// TwinCAT 3 PLC project PLC
// ProgramVersion: 3.1.4026.13
// CompilerDefines: VISU_USEPROPERTYINFO
// libraries:
//   Tc2_Standard, * (Beckhoff Automation GmbH)
//   Tc2_System, * (Beckhoff Automation GmbH)
//   VisuSymbols, 4.5.0.0 (System)
// project tree:
//   FBs/Control/Function Blocks/ FB_Config.TcPOU, FB_Control.TcPOU, FB_DeadBand.TcPOU, FB_FeedForward.TcPOU, FB_PID.TcPOU
//   FBs/Control/Smart/ FB_FlowSharing.TcPOU, FB_Smart.TcPOU
//   FBs/Filtering/ FB_Filtering.TcPOU (not stored), ST_Filter.TcDUT (not stored)
//   FBs/Input/Function Blocks/ FB_JoystickInputScaling.TcPOU (not stored), FB_Normalize.TcPOU (not stored), FB_PositionInputScaling.TcPOU (not stored), FB_WinchDistance.TcPOU
//   FBs/Motion/Background/ FB_Clock.TcPOU, FB_FlowControl.TcPOU, FB_InitialPos.TcPOU (not stored), FB_Vel2Flow.TcPOU
//   FBs/Motion/ FB_Homing.TcPOU (not stored), FB_Ramp.TcPOU, FB_SineMotionRef.TcPOU, FB_Step.TcPOU
//   FBs/Output/ FB_OutputNormalizing.TcPOU
//   FBs/Truck/ G_Truck.TcGVL, P_Truck.TcPOU (not stored)
//   / GlobalTextList.TcGTLO, Measuring.TcTTO, PlcTask.TcTTO
//   GVLs/ENUMs/ E_AutoModes.TcDUT, E_HomingModes.TcDUT, E_ManuelModes.TcDUT, E_Modes.TcDUT (not stored), E_Motion.TcDUT
//   GVLs/ G_Enables.TcGVL, G_HMI.TcGVL, G_Homing.TcGVL, G_Inputs.TcGVL (not stored), G_Mode.TcGVL, G_OPC.TcGVL, G_Output.TcGVL (not stored), G_Parameters.TcGVL, G_Signals.TcGVL, G_Temp.TcGVL, ST_Signals.TcDUT
//   GVLs/Static/ G_Config.TcGVL, G_FilterConstants.TcGVL, G_Joystick.TcGVL, G_Winch.TcGVL
//   Programs/Background PRGs/ P_Clock.TcPOU, P_Config.TcPOU, P_DanielFiltering.TcPOU, P_Filtering.TcPOU (not stored), P_Convetions.TcPOU
//   Programs/Control/ P_Control.TcPOU, P_DeadBand.TcPOU, P_FeedForward.TcPOU, P_Motion.TcPOU, P_PID.TcPOU
//   Programs/IO/ P_Inputs.TcPOU, P_Output.TcPOU
//   Programs/ MAIN.TcPOU, P_HMI.TcPOU
//   Programs/Test/ P_SineTest.TcPOU
//   XML/ FB_Derivator.TcPOU, FB_LowpassFilter.TcPOU, G_Init.TcGVL, FB_Integrator.TcPOU
// real-time tasks:
//   TASK PlcTask: cycle T#10ms, priority 20, ADS port 350
//   TASK Measuring: cycle T#5ms, priority 21, ADS port 351
// I/O:
//   DEVICE Device 1 (EtherCAT), AmsNetId 5.76.250.97.2.1
//     Term 1 (EK1200) [EK1200-5000 EtherCAT Power supply (2A E-Bus)]
//       Term 2 (EL1008) [EL1008 8Ch. Dig. Input 24V, 3ms]
//       Term 3 (EL2008) [EL2008 8Ch. Dig. Output 24V, 0.5A]
//       Term 4 (EL4032) [EL4032 2Ch. Ana. Output +/-10V, 12bit]
//       Term 5 (EL9011) [EL9011 End Terminal]
//   DEVICE Device 3 (EtherCAT) (disabled), AmsNetId 5.76.250.97.4.1
//     Term 6 (EK1818) [EK1818 EtherCAT IO-Coupler  (1A E-Bus, 8 Ch. Dig. In, 3ms, 4 Ch. Dig. Out 24V, 0,5A)]
//       Term 7 (EL3068) [EL3068 8Ch. Ana. Input 0-10V]
//       Term 8 (EL3068) [EL3068 8Ch. Ana. Input 0-10V]
//       Term 9 (EL3068) [EL3068 8Ch. Ana. Input 0-10V]
//       Term 10 (EL3068) [EL3068 8Ch. Ana. Input 0-10V]
//       Term 11 (EL4008) [EL4008 8Ch. Ana. Output 0-10V, 12bit]
//       Term 12 (EL4004) [EL4004 4Ch. Ana. Output 0-10V, 12bit]
//       Term 10 (EL9011) [EL9011 End Terminal]
//     Box 13 (Fraba EtherCAT) [Absolute Rotary Encoder IXARC V01.05]
//     Box 14 (Fraba EtherCAT) [Absolute Rotary Encoder IXARC V01.05]
// variable links:
//   PLC/PLC Instance <-> Device 1 (EtherCAT)/Term 1 (EK1200)/Term 2 (EL1008)
//     Measuring Inputs/G_Inputs.bErrorOne <-> Channel 3/Input
//     Measuring Inputs/G_Inputs.bErrorTwo <-> Channel 4/Input
//   PLC/PLC Instance <-> Device 1 (EtherCAT)/Term 1 (EK1200)/Term 3 (EL2008)
//     Measuring Outputs/G_Output.bEnableRelay <-> Channel 3/Output
//     PlcTask Outputs/G_Output.bEnableValveOne <-> Channel 1/Output
//     PlcTask Outputs/G_Output.bEnableValveTwo <-> Channel 2/Output
//   PLC/PLC Instance <-> Device 1 (EtherCAT)/Term 1 (EK1200)/Term 4 (EL4032)
//     PlcTask Outputs/G_Output.nValveOneOutput <-> AO Outputs Channel 2/Analog output
//     PlcTask Outputs/G_Output.nValveTwoOutput <-> AO Outputs Channel 1/Analog output
//   PLC/PLC Instance <-> Device 3 (EtherCAT)/Box 13 (Fraba EtherCAT)
//     Measuring Inputs/G_Inputs.nRawWinchEncoder <-> Encoder/Position Value
//   PLC/PLC Instance <-> Device 3 (EtherCAT)/Term 6 (EK1818)
//     Measuring Inputs/G_Inputs.bEnableButton <-> Channel 2/Input
//   PLC/PLC Instance <-> Device 3 (EtherCAT)/Term 6 (EK1818)/Term 11 (EL4008)
//     Measuring Outputs/G_Output.nExtrudeOutput <-> AO Outputs Channel 5/Analog output
//     Measuring Outputs/G_Output.nJibOutput <-> AO Outputs Channel 4/Analog output
//     Measuring Outputs/G_Output.nMainOutput <-> AO Outputs Channel 3/Analog output
//     Measuring Outputs/G_Output.nSlewOutput <-> AO Outputs Channel 2/Analog output
//     Measuring Outputs/G_Output.nWinchOutput <-> AO Outputs Channel 1/Analog output
//   PLC/PLC Instance <-> Device 3 (EtherCAT)/Term 6 (EK1818)/Term 7 (EL3068)
//     Measuring Inputs/G_Inputs.nRawJibPistonPosition <-> AI Standard Channel 8/Value
//     Measuring Inputs/G_Inputs.nRawJoystickExtrude <-> AI Standard Channel 5/Value
//     Measuring Inputs/G_Inputs.nRawJoystickJib <-> AI Standard Channel 3/Value
//     Measuring Inputs/G_Inputs.nRawJoystickMain <-> AI Standard Channel 4/Value
//     Measuring Inputs/G_Inputs.nRawJoystickRotation <-> AI Standard Channel 2/Value
//     Measuring Inputs/G_Inputs.nRawJoystickWinch <-> AI Standard Channel 1/Value
//     Measuring Inputs/G_Inputs.nRawMainPistonPosition <-> AI Standard Channel 7/Value
//   PLC/PLC Instance <-> Device 3 (EtherCAT)/Term 6 (EK1818)/Term 8 (EL3068)
//     Measuring Inputs/G_Inputs.nRawMainPaCyl <-> AI Standard Channel 6/Value
//     Measuring Inputs/G_Inputs.nRawMainPaDCV <-> AI Standard Channel 4/Value
//     Measuring Inputs/G_Inputs.nRawMainPbDCV <-> AI Standard Channel 5/Value
//     Measuring Inputs/G_Inputs.nRawSupplyPs <-> AI Standard Channel 7/Value
//   PLC/PLC Instance <-> Device 3 (EtherCAT)/Term 6 (EK1818)/Term 9 (EL3068)
//     Measuring Inputs/G_Inputs.nRawJibPaCyl <-> AI Standard Channel 3/Value
//     Measuring Inputs/G_Inputs.nRawJibPaDCV <-> AI Standard Channel 6/Value
//     Measuring Inputs/G_Inputs.nRawJibPbCyl <-> AI Standard Channel 4/Value
//     Measuring Inputs/G_Inputs.nRawJibPbDCV <-> AI Standard Channel 5/Value

CONFIGURATION PLC
    RESOURCE PLC ON TwinCAT3
        TASK Measuring(INTERVAL := T#5ms, PRIORITY := 21);
        TASK PlcTask(INTERVAL := T#10ms, PRIORITY := 20);
        PROGRAM P_Inputs WITH Measuring : P_Inputs;
        PROGRAM P_DanielFiltering WITH Measuring : P_DanielFiltering;
        PROGRAM P_Filtering WITH Measuring : P_Filtering;
        PROGRAM MAIN WITH PlcTask : MAIN;
    END_RESOURCE
END_CONFIGURATION

// ---- GVLs/ENUMs/E_AutoModes.TcDUT
{attribute 'qualified_only'}
{attribute 'strict'}
{attribute 'to_string'}
TYPE E_AutoModes :
(
	Normal,
	FlowSharing,
	Smart
);
END_TYPE

// ---- GVLs/ENUMs/E_HomingModes.TcDUT
{attribute 'qualified_only'}
{attribute 'strict'}
{attribute 'to_string'}
TYPE E_HomingModes :
(
	Off,	
	MainTest1,
	MainTest2,
	JibTest1,
	JibTest2,
	DualTest1,
	DualTest2,
	DualTest3,
	DualTest4
);
END_TYPE

// ---- GVLs/ENUMs/E_ManuelModes.TcDUT
{attribute 'qualified_only'}
{attribute 'strict'}
{attribute 'to_string'}
TYPE E_ManuelModes :
(
	ManDirect,
	ManConst,
	ManSpeed
);
END_TYPE

// ---- GVLs/ENUMs/E_Motion.TcDUT
{attribute 'qualified_only'}
{attribute 'strict'}
{attribute 'to_string'}
TYPE E_Motion :
(
	Sine,
	Ramp
);
END_TYPE

// ---- GVLs/ST_Signals.TcDUT
TYPE ST_Signals :
STRUCT
	fOutSignal 				: LREAL; // Signal Sent Out
	fOutCompansated			: LREAL; // DB Compansated, NOT IN USE
	fFF						: LREAL; // FeedForward Signal
	fPID					: LREAL; // PID Signal
	fError					: LREAL; // Signal Error
	fU						: LREAL; // FF + PID + DB
	fUAdj					: LREAL; // Adjusted U, for flow sharing
END_STRUCT
END_TYPE

// ---- FBs/Truck/G_Truck.TcGVL
{attribute 'qualified_only'}
VAR_GLOBAL
	bParked 		: BOOL;
	bDriveOut		: BOOL;
	fDriveOutTime	: LREAL;
	fTruckPosition 	: LREAL;
END_VAR

// ---- GVLs/G_Enables.TcGVL
{attribute 'qualified_only'}
VAR_GLOBAL
		
	bEmergencyButton 	: BOOL;

	bEnableU 			: BOOL;
	bEnableFF 			: BOOL;
	bEnablePID 			: BOOL;
	bEnableFlowShare	: BOOL;
	
	bEnableOne			: BOOL;
	bEnableTwo			: BOOL;
	bEnableThree		: BOOL;	
	
	bHoldButton 		: BOOL;
	
	bErrorOne 			: BOOL;
	bErrorTwo			: BOOL;
	bErrorThree			: BOOL;
	
	bSineMotion			: BOOL;
	bRampMotion			: BOOL;
	bRampAxis			: BOOL;
	bHoming				: BOOL;
	
	// Modes
	bAuto				: BOOL;
	bManual				: BOOL;
	bManDirect			: BOOL;
	bManConst			: BOOL;
	bManSpeed			: BOOL;
	
	// Config Enables
	bConfigJoysticks	: BOOL;
END_VAR

// ---- GVLs/G_HMI.TcGVL
{attribute 'qualified_only'}
VAR_GLOBAL
	// Mode Select
	nCounter				: INT;
	nHomingMode				: INT;
	nManuelMode				: INT;
	nAutoMode				: INT;
	nMotionMode				: INT;
	
	// Value Inputs
	fNumPad1				: LREAL;
	fNumPad2				: LREAL;
	
	// HMI Buttons
	bHoldButton_HMI			: BOOL;
	bstepp_button			: BOOL;
	bButton_Cylinder_1		: BOOL;
	bButton_Cylinder_2		: BOOL;
	bFlowShare				: BOOL;
	
END_VAR

// ---- GVLs/G_Homing.TcGVL
{attribute 'qualified_only'}
VAR_GLOBAL CONSTANT
	nArrLen 		: SINT := 7;
	//Variable  	: ARRAY[0..nArrLen] OF LREAL := [Main1, Main2, Jib1 , Jib2 , Dual1, Dual2, Dual3, Dual4];
	aHomingMain 	: ARRAY[0..nArrLen] OF LREAL := [0.300, 0.500, 0.500, 0.730, 0.500, 0.450, 0.700, 0.700]; // Main Position for tests
	aHomingJib 		: ARRAY[0..nArrLen] OF LREAL := [0.825, 0.080, 0.070, 0.250, 0.080, 0.380, 0.750, 0.050]; //  Jib Position for tests
	aHomingWinch 	: ARRAY[0..nArrLen] OF LREAL := [0.000, 0.000, 0.000, 0.000, 0.000, 0.000, 0.000, 0.000]; //Winch Position for tests
	aMinDistWinch	: ARRAY[0..nArrLen+1] OF LREAL := [-2,-2.50, -2.05, -2.05, -2.40, -2.05, -2.40, -2.80, -2.30]; //Winch Min Length
	aMaxDistWinch	: ARRAY[0..nArrLen+1] OF LREAL := [-10,-3.65, -2.60, -2.65, -5.05, -2.65, -2.75, -8.45, -3.60]; //Winch Max Length
	
	aNegMain		: ARRAY[0..nArrLen] OF BOOL := [FALSE, FALSE, FALSE, FALSE, FALSE, FALSE, TRUE , TRUE ];
	aNegJib			: ARRAY[0..nArrLen] OF BOOL := [FALSE, FALSE, FALSE, FALSE, FALSE, FALSE, TRUE , FALSE];
	aCosMain		: ARRAY[0..nArrLen] OF BOOL := [FALSE, FALSE, FALSE, FALSE, FALSE, FALSE, FALSE, FALSE];
	aCosJib			: ARRAY[0..nArrLen] OF BOOL := [FALSE, FALSE, FALSE, FALSE, FALSE, FALSE, FALSE, TRUE ];
	
	aMainMovement	: ARRAY[0..nArrLen] OF BOOL := [TRUE, TRUE, FALSE, FALSE, TRUE, TRUE, TRUE, TRUE];
	aJibMovement	: ARRAY[0..nArrLen] OF BOOL := [FALSE, FALSE, TRUE, TRUE, TRUE, TRUE, TRUE, TRUE];
END_VAR

// ---- GVLs/G_Mode.TcGVL
{attribute 'qualified_only'}
VAR_GLOBAL
	bAuto 		: BOOL;
	bManuel 	: BOOL;
	bRunning 	: BOOL;
END_VAR

// ---- GVLs/G_OPC.TcGVL
{attribute 'qualified_only'}
VAR_GLOBAL
	
	// System Values 
	fTime					: LREAL; // [s]
	nTime					: UINT;  // [s]
	fHoldTime				: LREAL; // [s]
	bMeasurement			: BOOL;
	fPs 					: ST_Filter; // [Bar]
	
	// MAIN Values
	fMainPaDCV				: ST_Filter; // [Bar]
	fMainPbDCV				: ST_Filter; // [Bar]
	fMainPaCyl				: ST_Filter; // [Bar]
	fMainPistonPosition 	: ST_Filter; // [m]
	fMainPistonVelocity		: LREAL; 	 // [m/s]
	fMainFlowA				: LREAL;	 // [L/min]
	fMainFlowB				: LREAL;	 // [L/min]
	
	// JIB Values
	fJibPaDCV				: ST_Filter; // [Bar]
	fJibPbDCV				: ST_Filter; // [Bar]
	fJibPaCyl				: ST_Filter; // [Bar]
	fJibPbCyl				: ST_Filter; // [Bar]
	fJibPistonPosition		: ST_Filter; // [m]
	fJibPistonVelocity		: LREAL; 	 // [m/s]
	fJibFlowA				: LREAL;	 // [L/min]
	fJibFlowB				: LREAL;	 // [L/min]
	
	// WINCH Values
	fWinchPa				: ST_Filter; // [Bar]
	fWinchPb				: ST_Filter; // [Bar]
	fWinchDistance			: ST_Filter; // [m]
	
	
	// Joystick Signals
	fJoystickWinch			: LREAL; // [-1, 1]
	fJoystickRotation		: LREAL; // [-1, 1]
	fJoystickMain			: LREAL; // [-1, 1]
	fJoystickJib			: LREAL; // [-1, 1]
	fJoystickExtrude		: LREAL; // [-1, 1]
	
	// Valve Signals
	fValveOneSignals		: ST_Signals; // [-1, 1]
	fValveTwoSignals		: ST_Signals; // [-1, 1]
	fFlowShareCoefficient	: LREAL;
	fFlowRef				: LREAL; // [L/min]
	
	// Motion Ref
	fMotionTime				: LREAL; // [s]
	fHomingTime				: LREAL; // [s]
	
	fXRefOne				: LREAL; // [m]
	fXDotRefOne				: LREAL; // [m/s]
	fFlowRefOne				: LREAL; // [L/min]
	fSmartFlowRefOne		: LREAL; // [L/min]
	fSmartVelRefOne			: LREAL; // [m/s]
	
	fXRefTwo				: LREAL; // [m]
	fXDotRefTwo				: LREAL; // [m/s]
	fFlowRefTwo				: LREAL; // [L/min]
	fSmartFlowRefTwo		: LREAL; // [L/min]
	fSmartVelRefTwo			: LREAL; // [m/s]
	
	fFlowPistonSide			: LREAL;
	fFlowRodSide			: LREAL;
	
END_VAR

// ---- GVLs/G_Parameters.TcGVL

{attribute 'qualified_only'}
VAR_GLOBAL
	
	// System Variable
	fTimeStep 			: LREAL := 0.010; // [s]
	
	fConst1 			: LREAL := 0.0; // [-1, 1]
	fConst2 			: LREAL := 0.0; // [-1, 1]
	
	fMaxFlow			: LREAL := 55.0; // [L/min]
	fRho				: LREAL := 850.0;
	fCd					: LREAL := 0.64;
	
	// Winch
	fMinWinchDist		: LREAL;
	fMaxWinchDist		: LREAL;
	
	// FeedForward Variables
	fOneMultiFF 		: LREAL := 1.0; // FeedForward Multipier
	fTwoMultiFF 		: LREAL := 1.0; // FeedForward Multipier
	
	// PID Variables
	fOneP 				: LREAL := 22.0; // P
	fOneI 				: LREAL := 0.0; // I
	fOneD 				: LREAL := 0.0; // D
		
	fTwoP 				: LREAL := 28.0; // P
	fTwoI 				: LREAL := 0.0; // I
	fTwoD 				: LREAL := 0.0; // D
	
	// Valve Variables
	// Valve 1 (Jib)
	fQMaxUpOne 			: LREAL := 20.0; // [L/min]
	fQMaxDownOne		: LREAL := 15.0; // [L/min]
	fDeltaP0One			: LREAL := 6.0; // [Bar]
	fDeadUpOne 			: LREAL := 0.037;
	fDeadDownOne		: LREAL := 0.111;
	fAreaUpOne			: LREAL := (fQMaxUpOne/6E4)/(fCd * SQRT(2/fRho * 6E5))*1E6; // [mm^2]
	fAreaDownOne		: LREAL := (fQMaxDownOne/6E4)/(fCd * SQRT(2/fRho * 6E5))*1E6; // [mm^2]
	
	// Valve 2 (Main)
	fQMaxUpTwo 			: LREAL := 20.0; // [L/min]
	fQMaxDownTwo		: LREAL := 15.0; // [L/min]
	fDeltaP0Two			: LREAL := 6.0; // [Bar]
	fDeadUpTwo 			: LREAL := 0.037;
	fDeadDownTwo		: LREAL := 0.105;
	fAreaUpTwo			: LREAL := (fQMaxUpTwo/6E4)/(fCd * SQRT(2/fRho * 6E5))*1E6;// [mm^2]
	fAreaDownTwo		: LREAL := (fQMaxDownTwo/6E4)/(fCd * SQRT(2/fRho * 6E5))*1E6;// [mm^2]
	
	// Piston Variables 
	fMaxStrokeMain 		: LREAL := 0.755; // [m]
	fMaxStrokeJib 		: LREAL := 0.856; // [m]

	fMaxSpeedMain		: LREAL := 0.1; // [m/s]
	fMaxSpeedJib		: LREAL := 0.1; // [m/s]
	
	aMaxFlowPist		: ARRAY[0..3] OF LREAL := [0.0 , 0.0 , 0.0 , 0.0]; 

	fDiaMain 			: LREAL := 160.0; // [mm]
	fDiaJib				: LREAL := 150.0; // [mm]
	fRodDiaMain			: LREAL := 100.0; // [mm]
	fRodDiaJib			: LREAL := 100.0; // [mm]
	
	fAreaMain			: LREAL := EXPT(fDiaMain/2 , 2) * Tc2_System.Global_Variables.PI/1E6; // [m^2]
	fAreaMainRod		: LREAL := (EXPT(fDiaMain/2 , 2)-EXPT(fRodDiaMain/2 , 2)) * Tc2_System.Global_Variables.PI/1E6; // [m^2]
	fAreaRelation1		: LREAL := fAreaMainRod / fAreaMain;

	fAreaJib			: LREAL := EXPT(fDiaJib/2 , 2) * Tc2_System.Global_Variables.PI / 1E6; // [m^2]
	fAreaJibRod			: LREAL := (EXPT(fDiaJib/2 , 2)- EXPT(fRodDiaJib/2 , 2)) * Tc2_System.Global_Variables.PI/1E6; // [m^2]
	fAreaRelation2		: LREAL := fAreaJibRod/fAreaJib;
	
	// MotionRef Variables
	fMainAmplitude 		: LREAL := 0.075; // [m]
	fMainFrequency		: LREAL := 1.0/40.0; // [Hz]
	
	fJibAmplitude		: LREAL := 0.1; // [m]
	fJibFrequency		: LREAL := 1.0/40.0; // [Hz]
	
	fRampConstStrJib	: LREAL := 0.4; // Signal Strength
	fRampConstStrMain	: LREAL := 0.3; // Signal Strength
	
	
END_VAR

// ---- GVLs/G_Signals.TcGVL
{attribute 'qualified_only'}
VAR_GLOBAL
	// MAIN Values
	fMainPaDCV				: ST_Filter; // [Bar]
	fMainPbDCV				: ST_Filter; // [Bar]
	fMainPaCyl				: ST_Filter; // [Bar]
	fMainPistonPosition 	: ST_Filter; // [m]
	
	// JIB Values
	fJibPaDCV				: ST_Filter; // [Bar]
	fJibPbDCV				: ST_Filter; // [Bar]
	fJibPaCyl				: ST_Filter; // [Bar]
	fJibPbCyl				: ST_Filter; // [Bar]
	fJibPistonPosition		: ST_Filter; // [m]
	
	// WINCH Values
	fWinchPa				: ST_Filter; // [Bar]
	fWinchPb				: ST_Filter; // [Bar]
	fWinchDistance			: ST_Filter; // [m]
END_VAR

// ---- GVLs/G_Temp.TcGVL
{attribute 'qualified_only'}
VAR_GLOBAL
	fRampJibIntegrated	: LREAL;
	fRampMainIntegrated	: LREAL;
END_VAR

// ---- GVLs/Static/G_Config.TcGVL
{attribute 'qualified_only'}
VAR_GLOBAL
	faMeasurement 			: ARRAY[0..100] OF LREAL;
	
	fJibJoystickAverage 	: LREAL;
	fConfigTime 			: LREAL;
	
	nArrayLength			: INT := 100;
	
	bJoystickConfig 		: BOOL;
END_VAR

// ---- GVLs/Static/G_FilterConstants.TcGVL
{attribute 'qualified_only'}
VAR_GLOBAL CONSTANT
	// Filter constants
	fPressureFilterNum 		: LREAL := 0.003137;
	fPressureFilterDenz 	: LREAL := 1.0;
	fPressureFilterDen 		: LREAL := -0.9969;
	fPressureFilterInit 	: LREAL := 0.0;
	
	fPosFilterNum 			: LREAL := 0.003137;
	fPosFilterDenz 			: LREAL := 1.0;
	fPosFilterDen 			: LREAL := -0.9969;
	fPosFilterInit 			: LREAL := 0.0;
	
	fSignalFilterNum 		: LREAL := 0.09516;
	fSignalFilterDenz 		: LREAL := 1.0;
	fSignalFilterDen 		: LREAL := -0.9048;
	fSignalFilterInit 		: LREAL := 0.0;
	
	fDerivatorFilterNum 	: LREAL := 0.0009995;
	fDerivatorFilterDenz 	: LREAL := 1.0;
	fDerivatorFilterDen 	: LREAL := -0.999;
	fDerivatorFilterInit 	: LREAL := 0.0;	
	
	fCutoffFreq             : LREAL := 0.0159; // 0.1;
    fDamping                : LREAL := 0.707106781186547;
	fSampleTime             : LREAL := 0.001;
END_VAR

// ---- GVLs/Static/G_Joystick.TcGVL
{attribute 'qualified_only'}
VAR_GLOBAL
	aMainCyl	: ARRAY[0..2] OF LREAL := [9650.0, 19369.0, 29152.0];
	aJibCyl		: ARRAY[0..2] OF LREAL := [9939.0, 19580.0, 28981.0];
	aWinch 		: ARRAY[0..2] OF LREAL := [9760.0, 19393.0, 28952.0];
	aRotation 	: ARRAY[0..2] OF LREAL := [9907.0, 19502.0, 29115.0];
	aExtrude 	: ARRAY[0..2] OF LREAL := [9939.0, 19640.0, 28916.0];
END_VAR

// ---- GVLs/Static/G_Winch.TcGVL
{attribute 'qualified_only'}
VAR_GLOBAL CONSTANT
	fStartPointPosition : LREAL := 0.0;
	fEndpointPosition 	: LREAL := 5.0;
    fStartPointValue 	: LREAL := 3803508.0;
	fEndPointValue 		: LREAL := 1556369.0;
END_VAR

// ---- XML/G_Init.TcGVL
VAR_GLOBAL CONSTANT
	SS_INITIALIZE	: SINT := 0;
	SS_STEP			: SINT := 1;
END_VAR

// ---- Programs/IO/P_Inputs.TcPOU
PROGRAM P_Inputs
VAR
	// Supply
	fbNormPs 					: FB_Normalize;
	
	// Main
	fbNormMainPaDCV				: FB_Normalize;
	fbNormMainPbDCV				: FB_Normalize;
	fbNormMainPaCyl 			: FB_Normalize;
	fbNormMainPistonPosition 	: FB_PositionInputScaling;
	
	// Jib
	fbNormJibPaDCV 				: FB_Normalize;
	fbNormJibPbDCV 				: FB_Normalize;
	fbNormJibPaCyl	 			: FB_Normalize;
	fbNormJibPbCyl	 			: FB_Normalize;
	fbNormJibPistonPosition 	: FB_PositionInputScaling;

	// Winch
	fbNormWinchPa 				: FB_Normalize;
	fbNormWinchPb 				: FB_Normalize;
	fbNormWinchEncoder			: FB_WinchDistance;

	// Joystick
	fbJoystickWinch 			: FB_JoystickInputScaling;
	fbJoystickRotation 			: FB_JoystickInputScaling;
	fbJoystickMain 				: FB_JoystickInputScaling;
	fbJoystickJib 				: FB_JoystickInputScaling;
	fbJoystickExtrude 			: FB_JoystickInputScaling;	
	
	fbWinchDistance				: FB_WinchDistance;
	
END_VAR

G_Enables.bEmergencyButton := G_Inputs.bEmergencySwitch;

IF G_Inputs.bEnableButton THEN
	G_Enables.bHoldButton := G_Inputs.bEnableButton;
ELSIF G_HMI.bHoldButton_HMI THEN
	G_Enables.bHoldButton := G_HMI.bHoldButton_HMI;
ELSE
	G_Enables.bHoldButton := FALSE;
END_IF

// Supply
fbNormPs(
	nRawInput := G_Inputs.nRawSupplyPs,
	fMaxValue := 400.0, 			// [Bar]
	fNormalizedInput => G_OPC.fPs.fSignal
);

// Main
fbNormMainPaDCV(
	nRawInput := G_Inputs.nRawMainPaDCV,
	fMaxValue := 400.0, 			// [Bar]
	fNormalizedInput => G_OPC.fMainPaDCV.fSignal
);

fbNormMainPbDCV(
	nRawInput := G_Inputs.nRawMainPbDCV,
	fMaxValue := 400.0, 			// [Bar]
	fNormalizedInput => G_OPC.fMainPbDCV.fSignal
);

fbNormMainPaCyl(
	nRawInput := G_Inputs.nRawMainPaCyl,
	fMaxValue := 400.0, 			// [Bar]
	fNormalizedInput => G_OPC.fMainPaCyl.fSignal
);

fbNormMainPistonPosition(
	nRawInput := G_Inputs.nRawMainPistonPosition,
	fMaxOutputValue := G_Parameters.fMaxStrokeMain,
	fMaxInputValue := 25990.0,
	fMinInputValue := 6639.0,
	fMinOutputValue := 0.081,
	fOffset := 0.0,
	fOutput => G_OPC.fMainPistonPosition.fSignal
);
	
// Jib
fbNormJibPaDCV(
	nRawInput := G_Inputs.nRawJibPaDCV,
	fMaxValue := 400.0, 			// [Bar]
	fNormalizedInput => G_OPC.fJibPaDCV.fSignal
);

fbNormJibPbDCV(
	nRawInput := G_Inputs.nRawJibPbDCV,
	fMaxValue := 400.0, 			// [Bar]
	fNormalizedInput => G_OPC.fJibPbDCV.fSignal
);

fbNormJibPaCyl(
	nRawInput := G_Inputs.nRawJibPaCyl,
	fMaxValue := 400.0, 			// [Bar]
	fNormalizedInput => G_OPC.fJibPaCyl.fSignal
);

fbNormJibPbCyl(
	nRawInput := G_Inputs.nRawJibPbCyl,
	fMaxValue := 400.0, 			// [Bar]
	fNormalizedInput => G_OPC.fJibPbCyl.fSignal
);

fbNormJibPistonPosition(
	nRawInput := G_Inputs.nRawJibPistonPosition,
	fMaxOutputValue := G_Parameters.fMaxStrokeJib,
	fMaxInputValue := 24925.0,
	fMinInputValue := 3065.0,
	fMinOutputValue := 0.0,
	fOffset := 0.0,
	fOutput => G_OPC.fJibPistonPosition.fSignal
);

// Winch
fbNormWinchPa(
	nRawInput := G_Inputs.nRawWinchPa,
	fMaxValue := 400.0, 			// [Bar]
	fNormalizedInput => G_OPC.fWinchPa.fSignal
);

fbNormWinchPb(
	nRawInput := G_Inputs.nRawWinchPb,
	fMaxValue := 400.0, 			// [Bar]
	fNormalizedInput => G_OPC.fWinchPb.fSignal
);

fbNormWinchEncoder(
	nWinchRaw := G_Inputs.nRawWinchEncoder,
	fWinchDistance => G_OPC.fWinchDistance.fSignal
);

// Joystick
fbJoystickWinch(
	nRawInput := G_Inputs.nRawJoystickWinch,
	bEnable := TRUE,
	fBitArray := G_Joystick.aWinch,
	fOutput => G_OPC.fJoystickWinch
);

fbJoystickRotation(
	nRawInput := G_Inputs.nRawJoystickRotation,
	bEnable := TRUE,
	fBitArray := G_Joystick.aRotation,
	fOutput => G_OPC.fJoystickRotation
);

fbJoystickMain(
	nRawInput := G_Inputs.nRawJoystickMain,
	bEnable := TRUE,
	fBitArray := G_Joystick.aMainCyl,
	fOutput => G_OPC.fJoystickMain
);

fbJoystickJib(
	nRawInput := G_Inputs.nRawJoystickJib,
	bEnable := TRUE,
	bInverse := TRUE,
	fBitArray := G_Joystick.aJibCyl,
	fOutput => G_OPC.fJoystickJib
);

fbJoystickExtrude(
	nRawInput := G_Inputs.nRawJoystickExtrude,
	bEnable := TRUE,
	fBitArray := G_Joystick.aExtrude,
	fOutput => G_OPC.fJoystickExtrude
);

END_PROGRAM

// ---- FBs/Input/Function Blocks/FB_WinchDistance.TcPOU
FUNCTION_BLOCK FB_WinchDistance
VAR_INPUT
	nWinchRaw : UDINT;
END_VAR
VAR_OUTPUT
	fWinchDistance : LREAL;
END_VAR
VAR
	fStartPointPosition : LREAL := 0.0;
	fEndpointPosition 	: LREAL := 5.0;
    fStartPointValue 	: LREAL := 3803508.0;
	fEndPointValue 		: LREAL := 1556369.0;
	fDxDu				: LREAL;
END_VAR

fDxDu := (fEndpointPosition - fStartPointPosition) / (fEndPointValue - fStartPointValue);
fWinchDistance:= -fDxDu*(TO_REAL(nWinchRaw) - fStartPointValue) + fStartPointPosition;

END_FUNCTION_BLOCK

// ---- Programs/Background PRGs/P_DanielFiltering.TcPOU
PROGRAM P_DanielFiltering
VAR
	fbFilterPs 					: FB_LowpassFilter;
	
	fbFilterMainPaDCV			: FB_LowpassFilter;
	fbFilterMainPbDCV			: FB_LowpassFilter;
	fbFilterMainPaCyl 			: FB_LowpassFilter;
	fbFilterMainPistonPosition 	: FB_LowpassFilter;
	fbFilterMainPistonVelocity	: FB_LowpassFilter;
	
	fbFilterJibPaDCV			: FB_LowpassFilter;
	fbFilterJibPbDCV			: FB_LowpassFilter;
	fbFilterJibPaCyl 			: FB_LowpassFilter;
	fbFilterJibPbCyl 			: FB_LowpassFilter;
	fbFilterJibPistonPosition 	: FB_LowpassFilter;
	fbFilterJibPistonVelocity	: FB_LowpassFilter;
	
	
	fbFilterWinchPa 			: FB_LowpassFilter;
	fbFilterWinchPb 			: FB_LowpassFilter;
	fbFilterWinchPosition		: FB_LowpassFilter;
	
	fbFilterU 					: FB_LowpassFilter;
END_VAR

// SUPPLY
fbFilterPs(
	fInput := G_OPC.fPs.fSignal,
	fDeltaT := G_FilterConstants.fSampleTime,
	fCutoffFreq := G_FilterConstants.fCutoffFreq,
	fDamping := G_FilterConstants.fDamping,
	
	fOutput => G_OPC.fPs.fDanielFilter
	
);

// MAIN
fbFilterMainPaDCV(
	fInput := G_OPC.fMainPaDCV.fSignal,
	fDeltaT := G_FilterConstants.fSampleTime,
	fCutoffFreq := G_FilterConstants.fCutoffFreq,
	fDamping := G_FilterConstants.fDamping,
	
	fOutput => G_OPC.fMainPaDCV.fDanielFilter
	
);

fbFilterMainPbDCV(
	fInput := G_OPC.fMainPbDCV.fSignal,
	fDeltaT := G_FilterConstants.fSampleTime,
	fCutoffFreq := G_FilterConstants.fCutoffFreq,
	fDamping := G_FilterConstants.fDamping,
	
	fOutput => G_OPC.fMainPbDCV.fDanielFilter
	
);

fbFilterMainPaCyl(
	fInput := G_OPC.fMainPaCyl.fSignal,
	fDeltaT := G_FilterConstants.fSampleTime,
	fCutoffFreq := G_FilterConstants.fCutoffFreq,
	fDamping := G_FilterConstants.fDamping,
	
	fOutput => G_OPC.fMainPaCyl.fDanielFilter
	
);

fbFilterMainPistonPosition(
	fInput := G_OPC.fMainPistonPosition.fSignal,
	fDeltaT := G_FilterConstants.fSampleTime,
	fCutoffFreq := G_FilterConstants.fCutoffFreq,
	fDamping := G_FilterConstants.fDamping,
	
	fOutput => G_OPC.fMainPistonPosition.fDanielFilter
	
);

fbFilterMainPistonVelocity(
	fInput:= G_OPC.fMainPistonPosition.fDanielFilter,
	fDeltaT := G_FilterConstants.fSampleTime,
	fCutoffFreq := G_FilterConstants.fCutoffFreq,
	fDamping := G_FilterConstants.fDamping,
	
	fOutput => G_OPC.fMainPistonPosition.fDanielFilter2
);

//JIB
fbFilterJibPaDCV(
	fInput := G_OPC.fJibPaDCV.fSignal,
	fDeltaT := G_FilterConstants.fSampleTime,
	fCutoffFreq := G_FilterConstants.fCutoffFreq,
	fDamping := G_FilterConstants.fDamping,
	
	fOutput => G_OPC.fJibPaDCV.fDanielFilter
	
);

fbFilterJibPbDCV(
	fInput := G_OPC.fJibPbDCV.fSignal,
	fDeltaT := G_FilterConstants.fSampleTime,
	fCutoffFreq := G_FilterConstants.fCutoffFreq,
	fDamping := G_FilterConstants.fDamping,
	
	fOutput => G_OPC.fJibPbDCV.fDanielFilter
	
);

fbFilterJibPaCyl(
	fInput := G_OPC.fJibPaCyl.fSignal,
	fDeltaT := G_FilterConstants.fSampleTime,
	fCutoffFreq := G_FilterConstants.fCutoffFreq,
	fDamping := G_FilterConstants.fDamping,
	
	fOutput => G_OPC.fJibPaCyl.fDanielFilter
	
);

fbFilterJibPbCyl(
	fInput := G_OPC.fJibPbCyl.fSignal,
	fDeltaT := G_FilterConstants.fSampleTime,
	fCutoffFreq := G_FilterConstants.fCutoffFreq,
	fDamping := G_FilterConstants.fDamping,
	
	fOutput => G_OPC.fJibPbCyl.fDanielFilter
	
);

fbFilterJibPistonPosition(
	fInput := G_OPC.fJibPistonPosition.fSignal,
	fDeltaT := G_FilterConstants.fSampleTime,
	fCutoffFreq := G_FilterConstants.fCutoffFreq,
	fDamping := G_FilterConstants.fDamping,
	
	fOutput => G_OPC.fJibPistonPosition.fDanielFilter	
);

fbFilterJibPistonVelocity(
	fInput:= G_OPC.fJibPistonPosition.fDanielFilter,
	fDeltaT := G_FilterConstants.fSampleTime,
	fCutoffFreq := G_FilterConstants.fCutoffFreq,
	fDamping := G_FilterConstants.fDamping,
	
	fOutput => G_OPC.fJibPistonPosition.fDanielFilter2
);

// WINCH
fbFilterWinchPa(
	fInput := G_OPC.fWinchPa.fSignal,
	fDeltaT := G_FilterConstants.fSampleTime,
	fCutoffFreq := G_FilterConstants.fCutoffFreq,
	fDamping := G_FilterConstants.fDamping,
	
	fOutput => G_OPC.fWinchPa.fDanielFilter
	
);

fbFilterWinchPb(
	fInput := G_OPC.fWinchPb.fSignal,
	fDeltaT := G_FilterConstants.fSampleTime,
	fCutoffFreq := G_FilterConstants.fCutoffFreq,
	fDamping := G_FilterConstants.fDamping,
	
	fOutput => G_OPC.fWinchPb.fDanielFilter
	
);

fbFilterWinchPosition(
	fInput := G_OPC.fWinchDistance.fSignal,
	fDeltaT := G_FilterConstants.fSampleTime,
	fCutoffFreq := G_FilterConstants.fCutoffFreq,
	fDamping := G_FilterConstants.fDamping,
	
	fOutput => G_OPC.fWinchDistance.fDanielFilter
	
);

END_PROGRAM

// ---- XML/FB_LowpassFilter.TcPOU
FUNCTION_BLOCK FB_LowpassFilter
VAR_INPUT
	fInput 				: LREAL;		      // Input
	fDeltaT				: LREAL; 			 // Cycle time [s]
	// Tuning Parameters 
	fCutoffFreq 		: LREAL := 0.5; 	  // seconds, value of 0 disables the filter
	fDamping 			: LREAL := 1/SQRT(2); // Damping ratio --> 0.707106781186547
	// Optional Parameters (Dont need to be used)
	bEnableLimits		: BOOL := FALSE;
	fLimitMax			: LREAL := 1.0;
	fLimitMin 			: LREAL := -1.0;
	// Optional Inputs (Dont need to be used)
	fDotInput_bypass 	: LREAL := 0;	      // Additional velocity input that bypasses the filter [unit/s]
	bReset 				: BOOL;				 // Resets the filter, and Sets Output = Input
END_VAR
VAR_OUTPUT
	fOutput 			: LREAL := fInput;	 // Output
	bError 				: BOOL;				 // TRUE if error
END_VAR
VAR
	fC 				: LREAL;
	fC2 			: LREAL; // c^2
	fDotOuptut 		: LREAL;
	fDot2Ouptut 	: LREAL;
	bFirstRun 		: BOOL := TRUE;
END_VAR

bError := FALSE;

IF (fCutoffFreq < 1E-10) THEN
	fOutput := fInput;
	bReset := TRUE;
END_IF

IF NOT bReset THEN
	fC := 2*PI*fDeltaT/fCutoffFreq;
	IF (fC <= 0) THEN
		bError := TRUE;
		bReset := TRUE;
	ELSIF (fC >= 0.9) THEN
		fC := 0.9;
	END_IF
END_IF

IF bReset OR bFirstRun THEN
	bFirstRun := FALSE;
	bReset := FALSE;
	fOutput := fInput;
	fDotOuptut  := 0;
	fDot2Ouptut := 0;
	RETURN;
END_IF

IF bError THEN RETURN; END_IF

fC2 := EXPT(fC, 2.0);

fDot2Ouptut := (fInput - fOutput)*fC2 - 2*fDamping*fC*fDotOuptut;

fDotOuptut := fDotOuptut + fDot2Ouptut;
fOutput := fOutput + fDotOuptut + fDotInput_bypass*fDeltaT;

IF ABS(fOutput) < 1E-10 THEN
	fOutput := 0;
END_IF

IF bEnableLimits THEN
	fOutput := LIMIT(fLimitMin,fOutput,fLimitMax);	
ELSE 
	fOutput := fOutput; 
END_IF

END_FUNCTION_BLOCK

// ---- Programs/MAIN.TcPOU
PROGRAM MAIN
VAR
	bTemp : BOOL;
END_VAR


P_Clock();
P_HMI();
P_DeadBand();
P_FeedForward();
P_PID();
P_Convetions();
P_Control();
P_Motion();
P_Output();
P_Truck();

// Test Programs
//P_SineTest();

END_PROGRAM

// ---- Programs/Background PRGs/P_Clock.TcPOU
PROGRAM P_Clock
VAR
	
	fbClock 		: FB_Clock;
	fbMotionClock 	: FB_Clock;
	fbDriveOut 		: FB_Clock;
	fbHoming		: FB_Clock;
	fbHoldTime		: FB_Clock;
	
END_VAR



fbClock(
	bStartEnable := G_HMI.bstepp_button,
	bEnableInt := G_HMI.bstepp_button,
	
	fTime => G_OPC.fTime,
	nTime => G_OPC.nTime
);

fbMotionClock(
	bStartEnable := (G_Enables.bSineMotion OR G_Enables.bRampMotion) AND G_Enables.bHoldButton AND G_Enables.bAuto, // AND G_HMI.bstepp_button AND G_Enables.bHoldButton,
	
	fTime => G_OPC.fMotionTime
);

fbDriveOut(
	bStartEnable := G_Truck.bDriveOut AND NOT(G_HMI.bstepp_button),
	
	fTime => G_Truck.fDriveOutTime
);

fbHoming(
	bStartEnable := G_HMI.bstepp_button AND G_Enables.bHoming,
	
	fTime => G_OPC.fHomingTime
);

fbHoldTime(
	bStartEnable := G_Enables.bHoldButton,
	
	fTime => G_OPC.fHoldTime
);

END_PROGRAM

// ---- FBs/Motion/Background/FB_Clock.TcPOU
FUNCTION_BLOCK FB_Clock
VAR_INPUT
	bStartEnable 	: BOOL;
	bEnableInt		: BOOL;
END_VAR
VAR_OUTPUT
	fTime 			: LREAL;
	nTime			: UINT;
END_VAR
VAR
END_VAR

IF NOT(bStartEnable) THEN
	fTime := 0.0;
	nTime := 0;
ELSE
	fTime := fTime + G_Parameters.fTimeStep;
END_IF

IF bEnableInt THEN
	nTime := LREAL_TO_UINT(fTime);
ELSE
	nTime := 0;
END_IF

END_FUNCTION_BLOCK

// ---- Programs/P_HMI.TcPOU
PROGRAM P_HMI
VAR
	fbDerivatorMainSpeed	: FB_Derivator;
	fbDerivatorJibSpeed		: FB_Derivator;
	fMainVelocity			: LREAL;
	fJibVelocity			: LREAL;

END_VAR

fbDerivatorMainSpeed(
	ssMethodType := 1,
	fSignal := G_OPC.fMainPistonPosition.fDanielFilter2,
	fSignalDerivative => fMainVelocity
);

fbDerivatorJibSpeed(
	ssMethodType := 1,
	fSignal := G_OPC.fJibPistonPosition.fDanielFilter2,
	fSignalDerivative => fJibVelocity
);

G_OPC.bMeasurement := G_HMI.bstepp_button;

IF fMainVelocity < -0.001 OR fMainVelocity > 0.001 THEN
	G_OPC.fMainPistonVelocity := fMainVelocity;
ELSE
	G_OPC.fMainPistonVelocity := 0.0;
END_IF

IF fJibVelocity < -0.001 OR fJibVelocity > 0.001 THEN
	G_OPC.fJibPistonVelocity := fJibVelocity;
ELSE
	G_OPC.fJibPistonVelocity := 0.0;
END_IF


IF G_HMI.nManuelMode < E_ManuelModes.ManDirect THEN
	G_HMI.nManuelMode := E_ManuelModes.ManDirect;
ELSIF G_HMI.nManuelMode > E_ManuelModes.ManSpeed THEN
	G_HMI.nManuelMode := E_ManuelModes.ManSpeed;
END_IF

IF G_HMI.nMotionMode < E_Motion.Sine THEN
	G_HMI.nMotionMode := E_Motion.Sine;
ELSIF G_HMI.nMotionMode > E_Motion.Ramp THEN
	G_HMI.nMotionMode := E_Motion.Ramp;
END_IF

IF G_HMI.nCounter < E_Modes.Manuel THEN
	G_HMI.nCounter := E_Modes.Manuel;
ELSIF G_HMI.nCounter > E_Modes.Auto THEN
	G_HMI.nCounter := E_Modes.Auto; 
END_IF

IF G_HMI.nAutoMode < E_AutoModes.Normal THEN
	G_HMI.nAutoMode := E_AutoModes.Normal;
ELSIF G_HMI.nAutoMode > E_AutoModes.Smart THEN
	G_HMI.nAutoMode := E_AutoModes.Smart;
END_IF

G_Parameters.fConst1 := G_HMI.fNumPad1;
G_Parameters.fConst2 := G_HMI.fNumPad2;

IF G_Enables.bErrorOne THEN
	G_Enables.bEnableOne := FALSE;
ELSE
	G_Enables.bEnableOne := G_Enables.bEnableOne;
END_IF

IF G_Enables.bErrorTwo THEN
	G_Enables.bEnableTwo := FALSE;
ELSE
	G_Enables.bEnableTwo := G_Enables.bEnableTwo;
END_IF

// IF G_Enables.bHoming THEN
// 	G_Enables.bEnablePID := FALSE;
// ELSE
// 	G_Enables.bEnablePID := G_Enables.bEnablePID;
// END_IF

IF G_HMI.nHomingMode < 0 THEN 
	G_HMI.nHomingMode := 0;
ELSIF G_HMI.nHomingMode > G_Homing.nArrLen + 1 THEN
	G_HMI.nHomingMode := G_Homing.nArrLen + 1;
ELSE
	G_HMI.nHomingMode := G_HMI.nHomingMode;
END_IF

END_PROGRAM

// ---- XML/FB_Derivator.TcPOU
FUNCTION_BLOCK FB_Derivator
VAR_INPUT
	ssMethodType		: SINT;
	fSignal				: LREAL;
END_VAR
VAR_OUTPUT
	fSignalDerivative	: LREAL;
END_VAR
VAR
	rtb_TSamp			: LREAL;
	UD_DSTATE			: LREAL;
END_VAR



CASE ssMethodType OF
    SS_INITIALIZE: 
        (* SystemInitialize for Atomic SubSystem: '<Root>/Derivator' *)
        (* InitializeConditions for UnitDelay: '<S2>/UD'
         *
         * Block description for '<S2>/UD':
         *  
         *  Store in Global RAM *)
        UD_DSTATE := 0.0;
        (* End of SystemInitialize for SubSystem: '<Root>/Derivator' *)
    SS_STEP: 
        (* Outputs for Atomic SubSystem: '<Root>/Derivator' *)
        (* SampleTimeMath: '<S2>/TSamp'
         *
         * About '<S2>/TSamp':
         *  y = u * K where K = 1 / ( w * Ts )
         *   *)
        rtb_TSamp := fSignal * 1000.0;
        (* Outport: '<Root>/fSignalDerivative' incorporates:
         *  Sum: '<S2>/Diff'
         *  UnitDelay: '<S2>/UD'
         *
         * Block description for '<S2>/Diff':
         *  
         *  Add in CPU
         *
         * Block description for '<S2>/UD':
         *  
         *  Store in Global RAM *)
        fSignalDerivative := rtb_TSamp - UD_DSTATE;
        (* Update for UnitDelay: '<S2>/UD'
         *
         * Block description for '<S2>/UD':
         *  
         *  Store in Global RAM *)
        UD_DSTATE := rtb_TSamp;
        (* End of Outputs for SubSystem: '<Root>/Derivator' *)
END_CASE;

END_FUNCTION_BLOCK

// ---- Programs/Control/P_DeadBand.TcPOU
PROGRAM P_DeadBand
VAR
	fbDeadBandOne : FB_DeadBand;
	fbDeadBandTwo : FB_DeadBand;
END_VAR

fbDeadBandOne(
	fSignal := G_OPC.fJoystickJib,
	fDeadBandUp := G_Parameters.fDeadUpOne,
	fDeadBanddown := G_Parameters.fDeadDownOne,
	fXDotRef := G_Parameters.fMaxSpeedMain * G_OPC.fJoystickJib,
	fCompansatedSignal =>G_OPC.fValveOneSignals.fOutCompansated
);

fbDeadBandTwo(
	fSignal := G_OPC.fJoystickMain,
	fDeadBandUp := G_Parameters.fDeadUpTwo,
	fDeadBanddown := G_Parameters.fDeadDownTwo,
	fXDotRef := G_Parameters.fMaxSpeedJib * G_OPC.fJoystickMain,
	fCompansatedSignal =>G_OPC.fValveTwoSignals.fOutCompansated
);

END_PROGRAM

// ---- FBs/Control/Function Blocks/FB_DeadBand.TcPOU
FUNCTION_BLOCK FB_DeadBand
VAR_INPUT
	fSignal : LREAL;
	fDeadBandUp : LREAL;
	fDeadBandDown : LREAL;
	fXDotRef : LREAL;
END_VAR
VAR_OUTPUT
	fCompansatedSignal : LREAL;
END_VAR
VAR
	fSignalUp : LREAL;
	fSignalDown : LREAL;
END_VAR

IF fXDotRef > 0 THEN
	fCompansatedSignal := fSignal + fDeadBandUp;
ELSIF fXDotRef < 0 THEN
	fCompansatedSignal := fSignal - fDeadBandDown;
ELSE
	fCompansatedSignal := 0.0;
END_IF

IF fCompansatedSignal < -1.0 THEN
	fCompansatedSignal := -1.0;
ELSIF fCompansatedSignal > 1.0 THEN
	fCompansatedSignal := 1.0;
ELSE
	fCompansatedSignal := fCompansatedSignal;
END_IF

END_FUNCTION_BLOCK

// ---- Programs/Control/P_FeedForward.TcPOU
PROGRAM P_FeedForward
VAR
	
	fbFFOne : FB_FeedForward;
	fbFFTwo : FB_FeedForward;
	
END_VAR

fbFFOne(
		fPs := G_OPC.fPs.fDanielFilter,
		fPa := G_OPC.fJibPaDCV.fDanielFilter,
		fPb := G_OPC.fJibPbDCV.fDanielFilter,
		
		fDeltaP0 := G_Parameters.fDeltaP0One,
		
		fMaxFlowUp := G_Parameters.fQMaxUpOne,
		fMaxFlowDown := G_Parameters.fQMaxDownOne,
		
		fDeadBandUp := G_Parameters.fDeadUpOne,
		fDeadBandDown := G_Parameters.fDeadDownOne,
		
		fArea := G_Parameters.fAreaJib,
		fPhi := G_Parameters.fAreaRelation2,
	);

	fbFFTwo(
		fPs := G_OPC.fPs.fDanielFilter,
		fPa := G_OPC.fMainPaDCV.fDanielFilter,
		fPb := G_OPC.fMainPbDCV.fDanielFilter,
		
		fDeltaP0 := G_Parameters.fDeltaP0Two,
		
		fMaxFlowUp := G_Parameters.fQMaxUpTwo,
		fMaxFlowDown := G_Parameters.fQMaxDownTwo,
		
		fDeadBandUp := G_Parameters.fDeadUpTwo,
		fDeadBandDown := G_Parameters.fDeadDownTwo,
		
		fArea := G_Parameters.fAreaMain,
		fPhi := G_Parameters.fAreaRelation1,
	); 

IF G_Enables.bAuto THEN
	fbFFOne(
		fXDot := G_OPC.fXDotRefOne,
		
		fUFF => G_OPC.fValveOneSignals.fFF,
		fFlow => G_OPC.fFlowRefOne
	);

	fbFFTwo(
		fXDot := G_OPC.fXDotRefTwo,
		
		fUFF => G_OPC.fValveTwoSignals.fFF,
		fFlow => G_OPC.fFlowRefTwo
	);
ELSIF G_Enables.bManual THEN
	fbFFOne(
		fXDot := G_OPC.fJoystickJib * G_Parameters.fMaxSpeedJib,
		
		fUFF => G_OPC.fValveOneSignals.fFF,
		fFlow => G_OPC.fFlowRefOne
	);

	fbFFTwo(
		fXDot := G_OPC.fJoystickMain * G_Parameters.fMaxSpeedMain,
		
		fUFF => G_OPC.fValveTwoSignals.fFF,
		fFlow => G_OPC.fFlowRefTwo
	);
END_IF

END_PROGRAM

// ---- FBs/Control/Function Blocks/FB_FeedForward.TcPOU
FUNCTION_BLOCK FB_FeedForward
VAR_INPUT
	fPs 			: LREAL; // [Bar]
	fPa 			: LREAL; // [Bar]
	fPb 			: LREAL; // [Bar]
	fXDot			: LREAL; // [m/s]
	fDeltaP0		: LREAL; // [Bar]
	fArea			: LREAL; // [mm^2]
	fPhi			: LREAL; // Relation between Areas
	fMaxFlowUp		: LREAL; // [L/min]
	fMaxFlowDown	: LREAL; // [L/min]
	fDeadBandUp		: LREAL; 
	fDeadBandDown	: LREAL;
END_VAR
VAR_OUTPUT
	fUFF 			: LREAL;
	fFlow			: LREAL; 	// Wanted Flow
END_VAR
VAR
	fSpoolTravel 	: LREAL; 	// Maximum Spool Travel
	fSlopeCharUp	: LREAL;	// Valve Slope Characteristic [mm/(L/min)]
	fSlopeCharDown	: LREAL;	// Valve Slope Characteristic [mm/(L/min)]
	fDeltaP_Norm	: LREAL; 	// Pressure Drop with Compansator
	
	
	fFlowLM			: LREAL;
	fDeltaP			: LREAL; 	// Pressure Drop
	fDeltaP_Ref		: LREAL; 	// Referance Pressure Drop
	fFlowRef		: LREAL; 	// Refereance Flow
	
	fUFFTemp		: LREAL;	// Temp Signal Out
END_VAR

fSpoolTravel 	:= 7.0; 								// Maximum Spool Travel
// fSlopeCharUp	:= (fSpoolTravel)/fMaxFlowUp; 			// Valve Slope Characteristic [mm/(L/min)]
// fSlopeCharDown	:= (fSpoolTravel)/fMaxFlowDown; 	// Valve Slope Characteristic [mm/(L/min)]
fDeltaP_Norm	:= fDeltaP0 * 100000.0;

IF fXDot > 0.0 THEN
	
	fFlow := fXDot * fArea;
	fFlowLM := fFlow * 60000;
	fDeltaP := (fPs - fPa) * 100000.0;
	IF fDeltaP < 100 THEN
		fDeltaP := 100;
	ELSE
		fDeltaP := fDeltaP;
	END_IF
	fDeltaP_Ref := ABS(fDeltaP_Norm/ (fDeltaP));
	fFlowRef := (fFlow * SQRT(fDeltaP_Ref)) * 60000.0;
	fUFFTemp := fFlowRef/fMaxFlowUp;
	fUFFTemp := fUFFTemp * (1.0-fDeadBandUp);
	
ELSIF fXDot < 0.0 THEN
	
	fFlow := fXDot * fArea * fPhi;
	fDeltaP := (fPs - fPb) * 100000.0;
	IF fDeltaP < 100 THEN
		fDeltaP := 100;
	ELSE
		fDeltaP := fDeltaP;
	END_IF
	fDeltaP_Ref := ABS(fDeltaP_Norm/(fDeltaP));
	fFlowRef := (fFlow * SQRT(fDeltaP_Ref)) * 60000.0;
	fUFFTemp := fFlowRef/fMaxFlowDown; //fUFFTemp :=	(fFlowRef * fSlopeCharDown) / fSpoolTravel;
	fUFFTemp := fUFFTemp*(1.0-fDeadBandDown);
	
ELSE
	
	fUFFTemp := 0.0;		

END_IF

IF fUFFTemp > 1.0 THEN
	fUFF := 1.0;
ELSIF fUFFTemp < -1.0 THEN
	fUFF := -1.0;
ELSE
	fUFF := fUFFTemp;
END_IF

END_FUNCTION_BLOCK

// ---- Programs/Control/P_PID.TcPOU
PROGRAM P_PID
VAR
	fbOnePID 				: FB_PID;
	fbTwoPID 				: FB_PID;
	fbIntegratorOne 		: FB_Integrator;
	fbDerivatorOne 			: FB_Derivator;
	fbDerivatorFilteringOne : FB_Filtering;
	fbIntegratorTwo 		: FB_Integrator;
	fbDerivatorTwo 			: FB_Derivator;
	fbDerivatorFilteringTwo : FB_Filtering;
END_VAR



IF G_Enables.bEnablePID AND NOT(G_Enables.bHoming) THEN
	// PID One
	fbDerivatorFilteringOne(
		ssMethodType := 1,
		Signal := fbOnePID.fSignalD,
		Num := G_FilterConstants.fDerivatorFilterNum,
		Denz := G_FilterConstants.fDerivatorFilterDenz,
		Den := G_FilterConstants.fDerivatorFilterDen,
		Initial := G_FilterConstants.fDerivatorFilterInit,
		Signal_Filtered => fbDerivatorOne.fSignal
	);
	
	fbIntegratorOne(
		ssMethodType := BOOL_TO_SINT(G_Enables.bHoldButton),
		fSignal := fbOnePID.fSignalI,
		fSignalIntegrated => fbOnePID.fSignalIntegrated
	);
	fbDerivatorOne(
		ssMethodType := BOOL_TO_SINT(G_Enables.bHoldButton),
		fSignal := fbOnePID.fSignalD,
		fSignalDerivative => fbOnePID.fSignalDerivated
	);

	fbOnePID(
		bEnablePID := G_Enables.bHoldButton AND G_Enables.bEnableOne ,
		fX := G_OPC.fXRefOne,
		fXReal := G_OPC.fJibPistonPosition.fDanielFilter,
		fKp := G_Parameters.fOneP,
		fKi := G_Parameters.fOneI,
		fKd := G_Parameters.fOneD,
		
		fError => G_OPC.fValveOneSignals.fError,
		fSignalAdjusted => G_OPC.fValveOneSignals.fPID
	);

	// PID Two
	fbDerivatorFilteringTwo(
		ssMethodType := 1,
		Signal := fbTwoPID.fSignalD,
		Num := G_FilterConstants.fDerivatorFilterNum,
		Denz := G_FilterConstants.fDerivatorFilterDenz,
		Den := G_FilterConstants.fDerivatorFilterDen,
		Initial := G_FilterConstants.fDerivatorFilterInit,
		Signal_Filtered => fbDerivatorTwo.fSignal
	);
	
	fbIntegratorTwo(
		ssMethodType := BOOL_TO_SINT(G_Enables.bHoldButton),
		fSignal := fbTwoPID.fSignalI,
		fSignalIntegrated => fbTwoPID.fSignalIntegrated
	);
	fbDerivatorTwo(
		ssMethodType := BOOL_TO_SINT(G_Enables.bHoldButton),
		fSignal := fbTwoPID.fSignalD,
		fSignalDerivative => fbTwoPID.fSignalDerivated
	);

	fbTwoPID(
		bEnablePID := G_Enables.bHoldButton AND G_Enables.bEnableTwo,
		fX := G_OPC.fXRefTwo,
		fXReal := G_OPC.fMainPistonPosition.fDanielFilter,
		fKp := G_Parameters.fTwoP,
		fKi := G_Parameters.fTwoI,
		fKd := G_Parameters.fTwoD,
		
		fError => G_OPC.fValveTwoSignals.fError,
		fSignalAdjusted => G_OPC.fValveTwoSignals.fPID
	);
	
ELSIF G_Enables.bEnablePID AND G_Enables.bHoming THEN
	
	// PID One
	fbDerivatorFilteringOne(
		ssMethodType := 1,
		Signal := fbOnePID.fSignalD,
		Num := G_FilterConstants.fDerivatorFilterNum,
		Denz := G_FilterConstants.fDerivatorFilterDenz,
		Den := G_FilterConstants.fDerivatorFilterDen,
		Initial := G_FilterConstants.fDerivatorFilterInit,
		Signal_Filtered => fbDerivatorOne.fSignal
	);
	
	fbIntegratorOne(
		ssMethodType := BOOL_TO_SINT(G_Enables.bHoming),
		fSignal := fbOnePID.fSignalI,
		fSignalIntegrated => fbOnePID.fSignalIntegrated
	);
	fbDerivatorOne(
		ssMethodType := BOOL_TO_SINT(G_Enables.bHoming),
		fSignal := fbOnePID.fSignalD,
		fSignalDerivative => fbOnePID.fSignalDerivated
	);

	fbOnePID(
		bEnablePID := G_Enables.bHoming AND G_Enables.bEnableOne ,
		fX := G_OPC.fXRefOne,
		fXReal := G_OPC.fJibPistonPosition.fDanielFilter,
		fKp := G_Parameters.fOneP,
		fKi := G_Parameters.fOneI,
		fKd := G_Parameters.fOneD,
		
		fError => G_OPC.fValveOneSignals.fError,
		fSignalAdjusted => G_OPC.fValveOneSignals.fPID
	);

	// PID Two
	fbDerivatorFilteringTwo(
		ssMethodType := 1,
		Signal := fbTwoPID.fSignalD,
		Num := G_FilterConstants.fDerivatorFilterNum,
		Denz := G_FilterConstants.fDerivatorFilterDenz,
		Den := G_FilterConstants.fDerivatorFilterDen,
		Initial := G_FilterConstants.fDerivatorFilterInit,
		Signal_Filtered => fbDerivatorTwo.fSignal
	);
	
	fbIntegratorTwo(
		ssMethodType := BOOL_TO_SINT(G_Enables.bHoming),
		fSignal := fbTwoPID.fSignalI,
		fSignalIntegrated => fbTwoPID.fSignalIntegrated
	);
	fbDerivatorTwo(
		ssMethodType := BOOL_TO_SINT(G_Enables.bHoming),
		fSignal := fbTwoPID.fSignalD,
		fSignalDerivative => fbTwoPID.fSignalDerivated
	);

	fbTwoPID(
		bEnablePID := G_Enables.bHoming AND G_Enables.bEnableTwo,
		fX := G_OPC.fXRefTwo,
		fXReal := G_OPC.fMainPistonPosition.fDanielFilter,
		fKp := G_Parameters.fTwoP,
		fKi := G_Parameters.fTwoI,
		fKd := G_Parameters.fTwoD,
		
		fError => G_OPC.fValveTwoSignals.fError,
		fSignalAdjusted => G_OPC.fValveTwoSignals.fPID
	);
	
END_IF

END_PROGRAM

// ---- FBs/Control/Function Blocks/FB_PID.TcPOU
FUNCTION_BLOCK FB_PID
VAR_INPUT
	bEnablePID			: BOOL;
	fX 					: LREAL;
	fXReal 				: LREAL;
	fSignalIntegrated 	: LREAL;
	fSignalDerivated 	: LREAL;
	fKp 				: LREAL;
	fKi 				: LREAL;
	fKd 				: LREAL;
END_VAR
VAR_OUTPUT
	fSignalI : LREAL;
	fSignalD : LREAL;
	fSignalAdjusted : LREAL;
	fError  : LREAL;
END_VAR
VAR
	fTempP : LREAL;
	fTempI : LREAL;
	fTempD : LREAL;
	fTempOut : LREAL;
END_VAR

fError := fX - fXReal;

// IF ABS(fError) < 0.0001 THEN
// 	fError := 0.0;	
// ELSE
// 	fError := fError;
// END_IF

fSignalI := fError;
fSignalD := fError;

fTempP := fError * fKp;
fTempI := fSignalIntegrated * fKi;
fTempD := fSignalDerivated * fKd;

fTempOut := fTempP + fTempI + fTempD;

IF fTempOut > 1.0 THEN
	fSignalAdjusted := 1.0;
ELSIF fTempOut < -1.0 THEN
	fSignalAdjusted := -1.0;
ELSE
	fSignalAdjusted := fTempOut;
END_IF

// IF ABS(fSignalAdjusted) < 1E-5 THEN
// 	fSignalAdjusted := 0.0;
// ELSE
// 	fSignalAdjusted := fSignalAdjusted;
// END_IF

IF bEnablePID THEN
	fSignalAdjusted := fSignalAdjusted;
ELSE
	fSignalAdjusted := 0.0;
END_IF

END_FUNCTION_BLOCK

// ---- XML/FB_Integrator.TcPOU
FUNCTION_BLOCK FB_Integrator
VAR_INPUT
	ssMethodType				: SINT;
	fSignal						: LREAL;
	nReset						: SINT;
END_VAR
VAR_OUTPUT
	fSignalIntegrated			: LREAL;
END_VAR
VAR
	c_DiscreteTimeIntegrator_Pr	: SINT;
	c_DiscreteTimeIntegrator_DS	: LREAL;
END_VAR



CASE ssMethodType OF
    SS_INITIALIZE: 
        (* SystemInitialize for Atomic SubSystem: '<Root>/Integrator' *)
        (* InitializeConditions for DiscreteIntegrator: '<S1>/Discrete-Time Integrator' *)
        c_DiscreteTimeIntegrator_DS := 0.0;
		c_DiscreteTimeIntegrator_Pr := 0;
        (* End of SystemInitialize for SubSystem: '<Root>/Integrator' *)
    SS_STEP: 
        (* Outputs for Atomic SubSystem: '<Root>/Integrator' *)
        (* Outport: '<Root>/fSignalIntegrated' incorporates:
         *  DiscreteIntegrator: '<S1>/Discrete-Time Integrator' *)
        IF (nReset <> 0.0) OR (c_DiscreteTimeIntegrator_Pr <> 0) THEN 
			c_DiscreteTimeIntegrator_DS := 0.0;
        END_IF;

		fSignalIntegrated := c_DiscreteTimeIntegrator_DS;
        (* Update for DiscreteIntegrator: '<S1>/Discrete-Time Integrator' *)
        c_DiscreteTimeIntegrator_DS := (0.01 * fSignal) + c_DiscreteTimeIntegrator_DS;
		
        IF nReset > 0.0 THEN 
             c_DiscreteTimeIntegrator_Pr := 1;
        ELSIF nReset < 0.0 THEN 
            c_DiscreteTimeIntegrator_Pr := -1;
        ELSIF nReset = 0.0 THEN 
             c_DiscreteTimeIntegrator_Pr := 0;
        ELSE 
             c_DiscreteTimeIntegrator_Pr := 2;
        END_IF;(* End of Outputs for SubSystem: '<Root>/Integrator' *)
END_CASE;

END_FUNCTION_BLOCK

// ---- Programs/Background PRGs/P_Convetions.TcPOU
PROGRAM P_Convetions
VAR
	fbMainVel2Flow	: FB_Vel2Flow;
	fbJibVel2Flow	: FB_Vel2Flow;
END_VAR

fbMainVel2Flow(
	fVelocity := G_OPC.fMainPistonVelocity,
	fArealUp := G_Parameters.fAreaMain,
	fArealDown := G_Parameters.fAreaMainRod,
	fXDotRef := G_OPC.fMainPistonVelocity,
	
	fFlowA => G_OPC.fMainFlowA,
	fFlowB => G_OPC.fMainFlowB
);

fbJibVel2Flow(
	fVelocity := G_OPC.fJibPistonVelocity,
	fArealUp := G_Parameters.fAreaJib,
	fArealDown := G_Parameters.fAreaJibRod,
	fXDotRef := G_OPC.fJibPistonVelocity,
	
	fFlowA => G_OPC.fJibFlowA,
	fFlowB => G_OPC.fJibFlowB
);

G_OPC.fFlowPistonSide := G_OPC.fJibFlowA + G_OPC.fMainFlowA;
G_OPC.fFlowRodSide := G_OPC.fJibFlowB + G_OPC.fMainFlowB;

END_PROGRAM

// ---- FBs/Motion/Background/FB_Vel2Flow.TcPOU
FUNCTION_BLOCK FB_Vel2Flow
VAR_INPUT
	fVelocity	: LREAL;
	fArealUp	: LREAL;
	fArealDown	: LREAL;
	fXDotRef	: LREAL;
END_VAR
VAR_OUTPUT
	fFlowA		: LREAL;
	fFlowB		: LREAL;
END_VAR
VAR
END_VAR

IF fXDotRef > 0.0 THEN
	fFlowA := fVelocity * fArealUp / 1E6 * 60000.0;
	fFlowB := fVelocity * fArealDown / 1E6 * 60000.0;
ELSIF fXDotRef < 0.0 THEN
	fFlowA := fVelocity * fArealUp / 1E6 * 60000.0;
	fFlowB := fVelocity * fArealDown / 1E6 * 60000.0;
ELSE
	fFlowA := 0.0;
	fFlowB := 0.0;
END_IF

END_FUNCTION_BLOCK

// ---- Programs/Control/P_Control.TcPOU
PROGRAM P_Control
VAR
	fbControl1 : FB_Control;
	fbControl2 : FB_Control;
END_VAR


IF G_Enables.bAuto THEN
	
	fbControl1(
		fFF := G_OPC.fValveOneSignals.fFF,
		fPID := G_OPC.fValveOneSignals.fPID,
		fDeadBandUp := G_Parameters.fDeadUpOne,
		fDeadBandDown := G_Parameters.fDeadDownOne,
		fKFF := G_Parameters.fOneMultiFF,

		bFF := G_Enables.bEnableFF,
		bPID := G_Enables.bEnablePID,
		bU := G_Enables.bEnableU,
		bValve := G_Enables.bEnableOne,
		bFlowShare := G_Enables.bEnableFlowShare, 
		
		fU => G_OPC.fValveOneSignals.fU,
		fUAdj => G_OPC.fValveOneSignals.fUAdj
	);
	
	fbControl2(
		fFF := G_OPC.fValveTwoSignals.fFF,
		fPID := G_OPC.fValveTwoSignals.fPID,
		fDeadBandUp := G_Parameters.fDeadUpTwo,
		fDeadBandDown := G_Parameters.fDeadDownTwo,
		fKFF := G_Parameters.fTwoMultiFF, 
		
		bFF := G_Enables.bEnableFF,
		bPID := G_Enables.bEnablePID,
		bU := G_Enables.bEnableU,
		bValve := G_Enables.bEnableTwo,
		bFlowShare := G_Enables.bEnableFlowShare,
		
		fU => G_OPC.fValveTwoSignals.fU,
		fUAdj => G_OPC.fValveTwoSignals.fUAdj
	);
	
ELSIF G_Enables.bManual THEN
	fbControl1(
		fFF := G_OPC.fValveOneSignals.fFF,
		fPID := G_OPC.fValveOneSignals.fPID,
		fDeadBandUp := G_Parameters.fDeadUpOne,
		fDeadBandDown := G_Parameters.fDeadDownOne,
		fKFF := G_Parameters.fOneMultiFF,

		bFF := G_Enables.bEnableFF,
		bPID := G_Enables.bEnablePID,
		bU := G_Enables.bEnableU, 
		
		fU => G_OPC.fValveOneSignals.fU
	);
	
	fbControl2(
		fFF := G_OPC.fValveTwoSignals.fFF,
		fPID := G_OPC.fValveTwoSignals.fPID,
		fDeadBandUp := G_Parameters.fDeadUpTwo,
		fDeadBandDown := G_Parameters.fDeadDownTwo,
		fKFF := G_Parameters.fTwoMultiFF, 
		
		bFF := G_Enables.bEnableFF,
		bPID := G_Enables.bEnablePID,
		bU := G_Enables.bEnableU,
		
		fU => G_OPC.fValveTwoSignals.fU
	);
	
ELSE
	G_OPC.fValveOneSignals.fU := 0.0;
	G_OPC.fValveTwoSignals.fU := 0.0;
END_IF

END_PROGRAM

// ---- FBs/Control/Function Blocks/FB_Control.TcPOU
FUNCTION_BLOCK FB_Control
VAR_INPUT
	fFF 			: LREAL;
	fPID			: LREAL;
	fDeadBandUp		: LREAL;
	fDeadBandDown	: LREAL;
	fKFF			: LREAL;
	fFlowSharing	: LREAL;
	
	bPID			: BOOL;
	bFF				: BOOL;
	bU				: BOOL;
	bValve			: BOOL;
	bFlowShare		: BOOL;
END_VAR
VAR_OUTPUT
	fU				: LREAL;
	fUAdj			: LREAL;
END_VAR
VAR
	FF				: LREAL;
	PID				: LREAL;
	fMaxOutput		: LREAL := 1.0;
END_VAR

IF bFlowShare THEN
	fFlowSharing := G_OPC.fFlowShareCoefficient;
ELSE
	fFlowSharing := 1.0;
END_IF

FF := fFF * fKFF * TO_INT(bFF);//* fMaxOutput;

PID := fPID * fMaxOutput * TO_INT(bPID);

fUAdj := (FF+PID)*TO_INT(bValve);

IF (fUAdj > 0.0) THEN
	fU := fUAdj*fFlowSharing + fDeadBandUp;
ELSIF (fUAdj < 0.0) THEN
	fU := fUAdj*fFlowSharing - fDeadBandDown;
ELSE
	fU := 0.0;
END_IF

IF fU < -1.0 THEN
	fU := -1.0;
ELSIF fU > 1.0 THEN
	fU := 1.0;
ELSE
	fU := fU;
END_IF

END_FUNCTION_BLOCK

// ---- Programs/Control/P_Motion.TcPOU
PROGRAM P_Motion
VAR
	fbSineMotionRefMain	: FB_SineMotionRef;
	fbSineMotionRefJib	: FB_SineMotionRef;
	
	fbRampMain			: FB_Ramp;
	fbRampJib			: FB_Ramp;

	fbHome	: FB_Homing;

	fbInitPosMain 		: FB_InitialPos;
	fbInitPosJib		: FB_InitialPos;
	
	fbIntegrator		: FB_Integrator;
	fbIntegratorMain	: FB_Integrator;
	fbIntegratorJib		: FB_Integrator;
	
	fbFlowShare			: FB_FlowSharing;
	fbSmart				: FB_Smart;
	
	bTest				: BOOL;
END_VAR

fbInitPosMain(
	bEnable := G_Enables.bHoldButton AND G_Enables.bEnableTwo,
	fCurrentPos := G_OPC.fMainPistonPosition.fDanielFilter
);

fbInitPosJib(
	bEnable := G_Enables.bHoldButton AND G_Enables.bEnableOne,
	fCurrentPos := G_OPC.fJibPistonPosition.fDanielFilter
);

fbSineMotionRefMain(
	fInitialPos := fbInitPosMain.fInitialPos,
	fTime := G_OPC.fMotionTime,
	fFrequency := G_Parameters.fMainFrequency,
	fAmplitude := G_Parameters.fMainAmplitude,
	fFlowShareCoff := fbFlowShare.fShareCoff
);

fbSineMotionRefJib(
	fInitialPos := fbInitPosJib.fInitialPos,
	fTime := G_OPC.fMotionTime,
	fFrequency := G_Parameters.fJibFrequency,
	fAmplitude := G_Parameters.fJibAmplitude,
	fFlowShareCoff := fbFlowShare.fShareCoff
);

fbRampMain(
	fTime := G_OPC.fMotionTime,
	fHeight := 0.01,
	fMaxSpeed := G_Parameters.fMaxSpeedMain
);

fbRampJib(
	fTime := G_OPC.fMotionTime,
	fHeight := 0.02,
	fMaxSpeed := G_Parameters.fMaxSpeedJib
);

G_Parameters.fMinWinchDist	:= ABS(G_Homing.aMinDistWinch[G_HMI.nHomingMode]);
G_Parameters.fMaxWinchDist	:= ABS(G_Homing.aMaxDistWinch[G_HMI.nHomingMode]);




IF G_HMI.bFlowShare THEN			
	fbFlowShare(
		fUAdjJib := G_OPC.fValveOneSignals.fUAdj,
		fUAdjMain := G_OPC.fValveTwoSignals.fUAdj,
		fMainAreaUp := G_Parameters.fAreaUpTwo,
		fMainAreaDown := G_Parameters.fAreaDownTwo,
		fJibAreaUp := G_Parameters.fAreaUpOne,
		fJibAreaDown := G_Parameters.fAreaDownOne,
		fCd := G_Parameters.fCd,
		fRho := G_Parameters.fRho,
		fMaxFlow := G_Parameters.fMaxFlow,
		fMainPa := G_OPC.fMainPaDCV.fDanielFilter,
		fMainPb := G_OPC.fMainPbDCV.fDanielFilter,
		fJibPa := G_OPC.fJibPaDCV.fDanielFilter,
		fJibPb := G_OPC.fJibPbDCV.fDanielFilter,
		fPs := G_OPC.fPs.fDanielFilter,
				
		fShareCoff => G_OPC.fFlowShareCoefficient,
		fFlowRef => G_OPC.fFlowRef
	);
ELSE
	G_OPC.fFlowShareCoefficient := 1.0;
END_IF

CASE G_HMI.nMotionMode OF
	E_Motion.Sine:
		G_Enables.bSineMotion := TRUE;
		G_Enables.bRampMotion := FALSE;
	E_Motion.Ramp:
		G_Enables.bSineMotion := FALSE;
		G_Enables.bRampMotion := TRUE;
END_CASE

IF G_Enables.bSineMotion AND NOT(G_Enables.bHoming) AND G_HMI.nHomingMode = 0 AND G_HMI.nMotionMode = 0 THEN
bTest := FALSE;
	fbIntegrator(
		ssMethodType := 1
	);
	
	fbSineMotionRefMain(
		bEnableMotion := G_Enables.bSineMotion AND G_Enables.bHoldButton AND G_Enables.bEnableTwo,
		
		fXDotRef => G_OPC.fXDotRefTwo,
		fXRef => G_OPC.fXRefTwo
	);
	
	fbSineMotionRefJib(
		bEnableMotion := G_Enables.bSineMotion AND G_Enables.bHoldButton AND G_Enables.bEnableOne,
		
		fXDotRef => G_OPC.fXDotRefOne,
		fXRef => G_OPC.fXRefOne
	);

ELSIF G_Enables.bRampMotion AND NOT(G_Enables.bHoming)  AND G_HMI.nMotionMode = 1 THEN

	IF G_Enables.bRampAxis THEN
		fbRampJib(
			bEnable := G_Enables.bRampMotion AND G_Enables.bHoldButton AND G_Enables.bEnableOne,
			fSignalStr := G_Parameters.fRampConstStrMain,
		
			fXDotRef => G_OPC.fXDotRefOne,
			fConst => G_OPC.fValveTwoSignals.fU
		);
		
		fbIntegratorJib(
			ssMethodType := TO_SINT(G_Enables.bRampMotion) * TO_SINT(G_OPC.fMotionTime > 0),
			fSignal := G_OPC.fXDotRefOne,
			fSignalIntegrated => G_Temp.fRampJibIntegrated
		);
		
		IF G_HMI.nHomingMode > 0 AND G_OPC.fMotionTime > 0 THEN
			G_OPC.fXRefOne := G_Homing.aHomingJib[G_HMI.nHomingMode - 1] + G_Temp.fRampJibIntegrated;
		END_IF
		
	ELSE
		
		fbRampMain(
			bEnable := G_Enables.bRampMotion AND G_Enables.bHoldButton AND G_Enables.bEnableTwo,
			fSignalStr := G_Parameters.fRampConstStrJib,
		
			fXDotRef => G_OPC.fXDotRefTwo,
			fConst => G_OPC.fValveOneSignals.fU
		);
		
		fbIntegratorMain(
			ssMethodType := TO_SINT(G_Enables.bRampMotion) * TO_SINT(G_OPC.fMotionTime > 0),
			fSignal := G_OPC.fXDotRefTwo,
			fSignalIntegrated => G_Temp.fRampMainIntegrated
		);
		
		IF G_HMI.nHomingMode > 0 AND G_OPC.fMotionTime > 0 THEN
			G_OPC.fXRefTwo := G_Homing.aHomingMain[G_HMI.nHomingMode - 1] + G_Temp.fRampMainIntegrated;
		END_IF
	END_IF
	
ELSIF G_Enables.bHoming AND NOT(G_Enables.bHoldButton) AND G_HMI.nHomingMode > 0 THEN
// Homing	
	fbHome(
		fWantedPositionMain := G_Homing.aHomingMain[G_HMI.nHomingMode - 1],
		fWantedPositionJib := G_Homing.aHomingJib[G_HMI.nHomingMode - 1],
		fCurrentPosMain := G_OPC.fMainPistonPosition.fDanielFilter,
		fCurrentPosJib := G_OPC.fJibPistonPosition.fDanielFilter,
		fClock := G_OPC.fHomingTime,
		bEnableHoming := G_Enables.bHoming,
		
		fXDotRefMain => G_OPC.fXDotRefTwo,
		fXDotRefJib => G_OPC.fXDotRefOne
	);
	
	G_OPC.fXRefOne := G_Homing.aHomingJib[G_HMI.nHomingMode - 1];
	G_OPC.fXRefTwo := G_Homing.aHomingMain[G_HMI.nHomingMode - 1];
	
ELSIF G_Enables.bHoldButton AND G_HMI.nHomingMode > 0 AND G_HMI.nMotionMode = 0 THEN
// Testing
	CASE G_HMI.nAutoMode OF
		E_AutoModes.Normal:
			
			G_Enables.bEnableOne := G_Homing.aJibMovement[G_HMI.nHomingMode - 1] AND G_Enables.bEnableThree;
			G_Enables.bEnableTwo := G_Homing.aMainMovement[G_HMI.nHomingMode - 1] AND G_Enables.bEnableThree;
			G_Enables.bEnableFlowShare := G_HMI.bFlowShare;
			
			fbSineMotionRefMain(
				bNegative := G_Homing.aNegMain[G_HMI.nHomingMode - 1],
				bCOS := G_Homing.aCosMain[G_HMI.nHomingMode - 1],
				bEnableMotion := G_Enables.bSineMotion AND G_Enables.bHoldButton AND G_Enables.bEnableTwo AND NOT(G_Enables.bHoming) AND G_Homing.aMainMovement[G_HMI.nHomingMode - 1],
			
				fXDotRef => G_OPC.fXDotRefTwo,
				fXRef => G_OPC.fXRefTwo
			);
					
			fbSineMotionRefJib(
				bNegative := G_Homing.aNegJib[G_HMI.nHomingMode - 1],
				bCOS := G_Homing.aCosJib[G_HMI.nHomingMode - 1],
				bEnableMotion := G_Enables.bSineMotion AND G_Enables.bHoldButton AND G_Enables.bEnableOne AND NOT(G_Enables.bHoming) AND G_Homing.aJibMovement[G_HMI.nHomingMode - 1],
				
				fXDotRef => G_OPC.fXDotRefOne,
				fXRef => G_OPC.fXRefOne
			);

			
		E_AutoModes.FlowSharing:
		
			G_Enables.bEnableOne := G_Homing.aJibMovement[G_HMI.nHomingMode - 1] AND G_Enables.bEnableThree;
			G_Enables.bEnableTwo := G_Homing.aMainMovement[G_HMI.nHomingMode - 1] AND G_Enables.bEnableThree;
			G_Enables.bEnableFlowShare := G_HMI.bFlowShare;
			
			fbSineMotionRefMain(
				bNegative := G_Homing.aNegMain[G_HMI.nHomingMode - 1],
				bCOS := G_Homing.aCosMain[G_HMI.nHomingMode - 1],
				bEnableMotion := G_Enables.bSineMotion AND G_Enables.bHoldButton AND G_Enables.bEnableTwo AND NOT(G_Enables.bHoming) AND G_Homing.aMainMovement[G_HMI.nHomingMode - 1],
			
				fXDotRef => G_OPC.fXDotRefTwo,
				fXRef => G_OPC.fXRefTwo
			);
					
			fbSineMotionRefJib(
				bNegative := G_Homing.aNegMain[G_HMI.nHomingMode - 1],
				bCOS := G_Homing.aCosMain[G_HMI.nHomingMode - 1],
				bEnableMotion := G_Enables.bSineMotion AND G_Enables.bHoldButton AND G_Enables.bEnableOne AND NOT(G_Enables.bHoming) AND G_Homing.aJibMovement[G_HMI.nHomingMode - 1],
				
				fXDotRef => G_OPC.fXDotRefOne,
				fXRef => G_OPC.fXRefOne
			);
			
	
	END_CASE
ELSE
	
	G_OPC.fXDotRefOne := 0.0;
	G_OPC.fXRefOne := G_OPC.fJibPistonPosition.fDanielFilter;
	
	G_OPC.fXDotRefTwo := 0.0;
	G_OPC.fXRefTwo := G_OPC.fMainPistonPosition.fDanielFilter;
	
	fbSineMotionRefMain(
		bEnableMotion := FALSE
		);
	fbSineMotionRefJib(
		bEnableMotion := FALSE
		);
END_IF

END_PROGRAM

// ---- FBs/Motion/FB_SineMotionRef.TcPOU
FUNCTION_BLOCK FB_SineMotionRef
VAR_INPUT
	bNegative : BOOL;
	bCOS : BOOL;
	fTime : LREAL;
	fAmplitude : LREAL;
	fFrequency : LREAL;
	fInitialPos : LREAL;
	bEnableMotion : BOOL;
	fFlowShareCoff : LREAL;
END_VAR
VAR_OUTPUT
	fXDotRef : LREAL;
	fXRef : LREAL;
END_VAR
VAR
	fXDotRefTemp : LREAL;
	fXRefTemp : LREAL;
	fMean : LREAL;
	fPeriod : LREAL;
	fPi : LREAL := Tc2_System.Global_Variables.PI;
	fDelta : LREAL;
END_VAR

fMean := fAmplitude + fInitialPos; 
IF ABS(fFrequency) > 0 THEN 
	fPeriod := 1 / fFrequency;
END_IF

IF bEnableMotion AND NOT(bCOS) THEN
	fXRefTemp := fMean - fAmplitude * COS(2 * fPi * fFrequency * fTime);
	fXDotRefTemp := 2 * fPi *fFrequency * fAmplitude * SIN(2* fPi * fFrequency * fTime);
ELSIF bEnableMotion AND bCOS THEN
	IF fTime < fPeriod / 4 THEN
		fXRefTemp := fInitialPos;
		fXDotRefTemp := 0.0;
	ELSIF fTime >= fPeriod / 4 THEN
		fXRefTemp := fMean - fAmplitude * COS(2 * fPi * fFrequency * (fTime-fPeriod/4) );
		fXDotRefTemp := 2 * fPi *fFrequency * fAmplitude * SIN(2* fPi * fFrequency * (fTime-fPeriod/4));
	END_IF
ELSE
	fXRefTemp := 0.0;
	fXDotRefTemp := 0.0;
END_IF 

fDelta := fInitialPos - fXRefTemp;

IF NOT(bNegative) AND NOT(bEnableMotion) THEN
	fXRef := fInitialPos;
	fXDotRef := 0.0;
ELSIF bNegative AND bEnableMotion THEN
	fXRef := fInitialPos + fDelta;
	fXDotRef := -fXDotRefTemp;
ELSE
	fXRef := fXRefTemp;
	fXDotRef := fXDotRefTemp;
END_IF

END_FUNCTION_BLOCK

// ---- FBs/Motion/FB_Ramp.TcPOU
FUNCTION_BLOCK FB_Ramp
VAR_INPUT
	bEnable 	: BOOL;

	fTime 		: LREAL;
	fMaxSpeed 	: LREAL;
	fHeight		: LREAL;
	
	fSignalStr	: LREAL;
END_VAR
VAR_OUTPUT
	fXDotRef 	: LREAL;
	fConst		: LREAL;
END_VAR
VAR
	fStartTime 	: LREAL := 1.0; // [s]
	fHoldTime 	: LREAL := 8.0; // [s]
	fRampTime 	: LREAL := 2.0; // [s]
	fSpeedRef	: LREAL;
	
	
	t1 			: LREAL;
	t2 			: LREAL;
	t3 			: LREAL;
	t35			: LREAL;
	t4 			: LREAL;
	t5 			: LREAL;
	t6 			: LREAL;
	t7 			: LREAL;
	t75			: LREAL;
	t8 			: LREAL;
	t9 			: LREAL;
END_VAR


fSpeedRef := fHeight/fRampTime;

IF fSpeedRef > fMaxSpeed THEN
    fSpeedRef := fMaxSpeed;
END_IF
 
t1  := fStartTime;
t2  := t1 + fRampTime;
t3  := t2 + fHoldTime/2;
t35 := t3 + fHoldTime/2;
t4  := t35 + fRampTime; 
t5  := t4 + fStartTime;
t6  := t5 + fRampTime;
t7  := t6 + fHoldTime/2; 
t75 := t7 + fHoldTime/2;
t8  := t75 + fRampTime;
t9  := t8 + fStartTime;

IF fTime = 0 THEN
	fXDotRef := 0.0;
	fConst := 0.0;
ELSIF fTime < t1 THEN // Start Delay
	fXDotRef := 0.0;
ELSIF fTime < t2 THEN // Ramp Up
	fXDotRef := -fSpeedRef * (fTime-t1);
ELSIF fTime < t3 THEN // Const Speed
	fXDotRef := -fSpeedRef * fRampTime;
ELSIF fTime < t35 THEN
	fXDotRef := -fSpeedRef * fRampTime;
	fConst := -fSignalStr;
ELSIF fTime < t4 THEN // Ramp Down
	fXDotRef := -fSpeedRef * fRampTime + fSpeedRef*(fTime-t35);
	fConst := 0.0;
ELSIF fTime < t5 THEN // Hold Time
	fXDotRef := 0.0;
ELSIF fTime < t6 THEN // Ramp Down
	fXDotRef := fSpeedRef * (fTime-t5);;
ELSIF fTime < t7 THEN // Const Speed
	fXDotRef := fSpeedRef * fRampTime;
ELSIF fTime < t75 THEN
	fXDotRef := fSpeedRef * fRampTime;
	fConst := fSignalStr;
ELSIF fTime < t8 THEN // Ramp Up
	fXDotRef := fSpeedRef * fRampTime - fSpeedRef * (fTime-t75);
	fConst := 0.0;
ELSIF fTime < t9 THEN // Stop
	fXDotRef := 0.0;
END_IF

END_FUNCTION_BLOCK

// ---- FBs/Control/Smart/FB_FlowSharing.TcPOU
FUNCTION_BLOCK FB_FlowSharing
VAR_INPUT
	fUAdjMain			: LREAL;
	fUAdjJib			: LREAL;
	fMainAreaUp			: LREAL;
	fMainAreaDown		: LREAL;
	fJibAreaUp			: LREAL;
	fJibAreaDown		: LREAL;
	fCd					: LREAL;
	fRho				: LREAL;
	fMaxFlow			: LREAL;
	fMainPa				: LREAL;
	fMainPb				: LREAL;
	fJibPa				: LREAL;
	fJibPb				: LREAL;
	fPs					: LREAL;
END_VAR
VAR_OUTPUT
	fShareCoff 			: LREAL;
	fFlowRef			: LREAL;
END_VAR
VAR
	fFlowRefSI			: LREAL;
	fDeltaPressure 		: LREAL;
	fKJib				: LREAL;
	fKMain				: LREAL;
	fFlowRefJib			: LREAL;
	fFlowRefMain		: LREAL;
END_VAR


IF fUAdjJib > 0 THEN
	
	fDeltaPressure := (fPs - fJibPa) * 1E5;
	
	IF fDeltaPressure <= 100 THEN
		fDeltaPressure := 100;
	END_IF
	
	fKJib := fJibAreaUp * 1E-6 * fCd * SQRT(2/fRho);
	fFlowRefJib := fKJib * fUAdjJib * SQRT(fDeltaPressure);
	
ELSIF fUAdjJib < 0 THEN
	
	fDeltaPressure := (fPs - fJibPb) * 1E5;
	
	IF fDeltaPressure <= 100 THEN
		fDeltaPressure := 100;
	END_IF
	
	fKJib :=fJibAreaDown * 1E-6 * fCd * SQRT(2/fRho);
	fFlowRefJib := fKJib * fUAdjJib * SQRT(fDeltaPressure);
	
ELSE
	
	fFlowRefJib := 0.0;
	
END_IF

IF fUAdjMain > 0 THEN
	
	fDeltaPressure := (fPs - fMainPa) * 1E5;
	
	IF fDeltaPressure <= 100 THEN
		fDeltaPressure := 100;
	END_IF
	
	fKMain := fMainAreaUp * 1E-6 * fCd * SQRT(2/fRho);
	fFlowRefMain := fKMain * fUAdjMain * SQRT(fDeltaPressure);
	
ELSIF fUAdjMain < 0 THEN
	
	fDeltaPressure := (fPs - fMainPb) * 1E5;
	
	IF fDeltaPressure <= 100 THEN
		fDeltaPressure := 100;
	END_IF
	
	fKMain := fMainAreaDown * 1E-6 * fCd * SQRT(2/fRho);
	fFlowRefMain := fKMain * fUAdjMain * SQRT(fDeltaPressure);
	
ELSE
	
	fFlowRefMain := 0.0;
	
END_IF

fFlowRefSI := (ABS(fFlowRefJib) + ABS(fFlowRefMain));
fFlowRef := (ABS(fFlowRefJib) + ABS(fFlowRefMain)) * 6E4;

IF fFlowRef <= 0.0 THEN
	fShareCoff := 1.0;
ELSE
	fShareCoff := fMaxFlow/fFlowRef;
END_IF

IF fShareCoff > 1.0 THEN
	fShareCoff := 1.0;
ELSIF fShareCoff < 0.0 THEN
	fShareCoff:= 0.0;
ELSE 
	fShareCoff := fShareCoff;
END_IF

END_FUNCTION_BLOCK

// ---- FBs/Control/Smart/FB_Smart.TcPOU
FUNCTION_BLOCK FB_Smart
VAR_INPUT
END_VAR
VAR_OUTPUT
END_VAR
VAR
END_VAR

END_FUNCTION_BLOCK

// ---- Programs/IO/P_Output.TcPOU
PROGRAM P_Output
VAR
	Mode : E_Modes;
	ManModes : E_ManuelModes;
	fbStepMain : FB_Step;
	fbStepJib : FB_Step;
END_VAR

IF INT_TO_LREAL(G_Output.nValveOneOutput)/32767.0 > 0 THEN
	G_OPC.fValveOneSignals.fOutSignal := INT_TO_LREAL(G_Output.nValveOneOutput)/32767.0 - G_Parameters.fDeadUpOne;
ELSIF INT_TO_LREAL(G_Output.nValveOneOutput)/32767.0 < 0 THEN
	G_OPC.fValveOneSignals.fOutSignal := INT_TO_LREAL(G_Output.nValveOneOutput)/32767.0 + G_Parameters.fDeadDownOne;
ELSE
	G_OPC.fValveOneSignals.fOutSignal := 0.0;
END_IF

IF INT_TO_LREAL(G_Output.nValveTwoOutput)/32767.0 > 0 THEN
	G_OPC.fValveTwoSignals.fOutSignal := INT_TO_LREAL(G_Output.nValveTwoOutput)/32767.0 - G_Parameters.fDeadUpTwo;
ELSIF INT_TO_LREAL(G_Output.nValveTwoOutput)/32767.0 < 0 THEN
	G_OPC.fValveTwoSignals.fOutSignal := INT_TO_LREAL(G_Output.nValveTwoOutput)/32767.0 + G_Parameters.fDeadDownTwo;
ELSE
	G_OPC.fValveTwoSignals.fOutSignal := 0.0;
END_IF

IF G_Enables.bHoldButton OR G_Enables.bHoming THEN
	CASE G_HMI.nCounter OF
		
		E_Modes.Manuel:
		
			G_Enables.bAuto := FALSE;
			G_Enables.bManual := TRUE;
		
			CASE G_HMI.nManuelMode OF
					
				E_ManuelModes.ManDirect:
				
					G_Output.bEnableValveOne := G_Enables.bHoldButton AND G_Enables.bEnableOne AND NOT(G_Enables.bErrorOne);
					G_Output.bEnableValveTwo := G_Enables.bHoldButton AND G_Enables.bEnableTwo AND NOT(G_Enables.bErrorTwo);
					G_Output.nValveOneOutput := LREAL_TO_INT(G_OPC.fJoystickMain * 32767.0);
					G_Output.nValveTwoOutput := LREAL_TO_INT(G_OPC.fJoystickJib * 32767.0);
					G_Enables.bManConst := FALSE;
					G_Enables.bManSpeed := FALSE;
					G_Enables.bManDirect := TRUE;
					
				E_ManuelModes.ManConst:
				
					G_Output.bEnableValveOne := G_Enables.bHoldButton AND G_Enables.bEnableOne AND NOT(G_Enables.bErrorOne);
					G_Output.bEnableValveTwo := G_Enables.bHoldButton AND G_Enables.bEnableTwo AND NOT(G_Enables.bErrorTwo);
					G_Output.nValveOneOutput := LREAL_TO_INT(G_Parameters.fConst1 * 32767.0);
					G_Output.nValveTwoOutput := LREAL_TO_INT(G_Parameters.fConst2 * 32767.0);
					G_Enables.bManDirect := FALSE;
					G_Enables.bManSpeed := FALSE;
					G_Enables.bManConst := TRUE;
					
				E_ManuelModes.ManSpeed:
					
					fbStepMain(
						bEnable := G_Enables.bHoldButton AND G_Enables.bEnableTwo,
						fSignal := G_Parameters.fConst2,
						
						fOutput => G_OPC.fValveTwoSignals.fU
					);
					
					fbStepJib(
						bEnable := G_Enables.bHoldButton AND G_Enables.bEnableOne,
						fSignal := G_Parameters.fConst1,
						
						fOutput => G_OPC.fValveOneSignals.fU
					);
					
					G_Output.bEnableValveOne := G_Enables.bHoldButton AND G_Enables.bEnableOne AND NOT(G_Enables.bErrorOne);
					G_Output.bEnableValveTwo := G_Enables.bHoldButton AND G_Enables.bEnableTwo AND NOT(G_Enables.bErrorTwo);
					G_Output.nValveOneOutput := LREAL_TO_INT(G_OPC.fValveOneSignals.fU * 32767.0) ;
					G_Output.nValveTwoOutput := LREAL_TO_INT(G_OPC.fValveTwoSignals.fU * 32767.0) ;
					G_Enables.bManDirect := FALSE;
					G_Enables.bManConst := FALSE;
					G_Enables.bManSpeed := TRUE;
					
				ELSE
				
					G_Enables.bManConst := FALSE;
					G_Enables.bManSpeed := FALSE;
					G_Enables.bManDirect := FALSE;
					
			END_CASE
			
		E_Modes.Off:
			G_Enables.bHoming := FALSE;
			G_Enables.bSineMotion := FALSE;
			G_Enables.bRampMotion := FALSE;
			G_Enables.bEnableOne := FALSE;
			G_Enables.bEnableTwo := FALSE;
			G_Enables.bAuto := FALSE;	
			G_Enables.bManual := FALSE;	

		E_Modes.Auto:
			
			CASE G_HMI.nHomingMode OF
				
				E_HomingModes.Off:
					G_Output.bEnableValveOne := G_Enables.bHoldButton AND G_Enables.bEnableOne AND NOT(G_Enables.bErrorOne);
					G_Output.bEnableValveTwo := G_Enables.bHoldButton AND G_Enables.bEnableTwo AND NOT(G_Enables.bErrorTwo);
					G_Output.nValveOneOutput := LREAL_TO_INT(G_OPC.fValveOneSignals.fU * 32767.0) * BOOL_TO_INT(G_Enables.bEnableU);
					G_Output.nValveTwoOutput := LREAL_TO_INT(G_OPC.fValveTwoSignals.fU * 32767.0) * BOOL_TO_INT(G_Enables.bEnableU);
					G_Enables.bManual := FALSE;
					G_Enables.bAuto := TRUE;
					
				E_HomingModes.MainTest1:
					G_Output.bEnableValveOne := (G_Enables.bHoldButton OR G_Enables.bHoming) AND G_Enables.bEnableOne AND NOT(G_Enables.bErrorOne);
					G_Output.bEnableValveTwo := (G_Enables.bHoldButton OR G_Enables.bHoming) AND G_Enables.bEnableTwo AND NOT(G_Enables.bErrorTwo);
					G_Output.nValveOneOutput := LREAL_TO_INT(G_OPC.fValveOneSignals.fU * 32767.0) ;
					G_Output.nValveTwoOutput := LREAL_TO_INT(G_OPC.fValveTwoSignals.fU * 32767.0) ;
					G_Enables.bManual := FALSE;
					G_Enables.bAuto := TRUE;
				
				E_HomingModes.MainTest2:
					G_Output.bEnableValveOne := (G_Enables.bHoldButton OR G_Enables.bHoming) AND G_Enables.bEnableOne AND NOT(G_Enables.bErrorOne);
					G_Output.bEnableValveTwo := (G_Enables.bHoldButton OR G_Enables.bHoming) AND G_Enables.bEnableTwo AND NOT(G_Enables.bErrorTwo);
					G_Output.nValveOneOutput := LREAL_TO_INT(G_OPC.fValveOneSignals.fU * 32767.0) ;
					G_Output.nValveTwoOutput := LREAL_TO_INT(G_OPC.fValveTwoSignals.fU * 32767.0) ;
					G_Enables.bManual := FALSE;
					G_Enables.bAuto := TRUE;
				
				E_HomingModes.JibTest1:
					G_Output.bEnableValveOne := (G_Enables.bHoldButton OR G_Enables.bHoming) AND G_Enables.bEnableOne AND NOT(G_Enables.bErrorOne);
					G_Output.bEnableValveTwo := (G_Enables.bHoldButton OR G_Enables.bHoming) AND G_Enables.bEnableTwo AND NOT(G_Enables.bErrorTwo);
					G_Output.nValveOneOutput := LREAL_TO_INT(G_OPC.fValveOneSignals.fU * 32767.0) ;
					G_Output.nValveTwoOutput := LREAL_TO_INT(G_OPC.fValveTwoSignals.fU * 32767.0) ;
					G_Enables.bManual := FALSE;
					G_Enables.bAuto := TRUE;
					
				E_HomingModes.JibTest2:
					G_Output.bEnableValveOne := (G_Enables.bHoldButton OR G_Enables.bHoming) AND G_Enables.bEnableOne AND NOT(G_Enables.bErrorOne);
					G_Output.bEnableValveTwo := (G_Enables.bHoldButton OR G_Enables.bHoming) AND G_Enables.bEnableTwo AND NOT(G_Enables.bErrorTwo);
					G_Output.nValveOneOutput := LREAL_TO_INT(G_OPC.fValveOneSignals.fU * 32767.0) ;
					G_Output.nValveTwoOutput := LREAL_TO_INT(G_OPC.fValveTwoSignals.fU * 32767.0) ;
					G_Enables.bManual := FALSE;
					G_Enables.bAuto := TRUE;
					
				E_HomingModes.DualTest1:
					G_Output.bEnableValveOne := (G_Enables.bHoldButton OR G_Enables.bHoming) AND G_Enables.bEnableOne AND NOT(G_Enables.bErrorOne);
					G_Output.bEnableValveTwo := (G_Enables.bHoldButton OR G_Enables.bHoming) AND G_Enables.bEnableTwo AND NOT(G_Enables.bErrorTwo);
					G_Output.nValveOneOutput := LREAL_TO_INT(G_OPC.fValveOneSignals.fU * 32767.0) ;
					G_Output.nValveTwoOutput := LREAL_TO_INT(G_OPC.fValveTwoSignals.fU * 32767.0) ;
					G_Enables.bManual := FALSE;
					G_Enables.bAuto := TRUE;
				
				E_HomingModes.DualTest2:
					G_Output.bEnableValveOne := (G_Enables.bHoldButton OR G_Enables.bHoming) AND G_Enables.bEnableOne AND NOT(G_Enables.bErrorOne);
					G_Output.bEnableValveTwo := (G_Enables.bHoldButton OR G_Enables.bHoming) AND G_Enables.bEnableTwo AND NOT(G_Enables.bErrorTwo);
					G_Output.nValveOneOutput := LREAL_TO_INT(G_OPC.fValveOneSignals.fU * 32767.0) ;
					G_Output.nValveTwoOutput := LREAL_TO_INT(G_OPC.fValveTwoSignals.fU * 32767.0) ;
					G_Enables.bManual := FALSE;
					G_Enables.bAuto := TRUE;;
					
				E_HomingModes.DualTest3:
					G_Output.bEnableValveOne := (G_Enables.bHoldButton OR G_Enables.bHoming) AND G_Enables.bEnableOne AND NOT(G_Enables.bErrorOne);
					G_Output.bEnableValveTwo := (G_Enables.bHoldButton OR G_Enables.bHoming) AND G_Enables.bEnableTwo AND NOT(G_Enables.bErrorTwo);
					G_Output.nValveOneOutput := LREAL_TO_INT(G_OPC.fValveOneSignals.fU * 32767.0) ;
					G_Output.nValveTwoOutput := LREAL_TO_INT(G_OPC.fValveTwoSignals.fU * 32767.0) ;
					G_Enables.bManual := FALSE;
					G_Enables.bAuto := TRUE;
					
				E_HomingModes.DualTest4:
					G_Output.bEnableValveOne := (G_Enables.bHoldButton OR G_Enables.bHoming) AND G_Enables.bEnableOne AND NOT(G_Enables.bErrorOne);
					G_Output.bEnableValveTwo := (G_Enables.bHoldButton OR G_Enables.bHoming) AND G_Enables.bEnableTwo AND NOT(G_Enables.bErrorTwo);
					G_Output.nValveOneOutput := LREAL_TO_INT(G_OPC.fValveOneSignals.fU * 32767.0) ;
					G_Output.nValveTwoOutput := LREAL_TO_INT(G_OPC.fValveTwoSignals.fU * 32767.0) ;
					G_Enables.bManual := FALSE;
					G_Enables.bAuto := TRUE;
								
			END_CASE
			
			
			
		ELSE
			G_Enables.bEnableOne := FALSE;
			G_Enables.bEnableTwo := FALSE;
			G_Enables.bAuto := FALSE;
			G_Enables.bManual := FALSE;
	END_CASE
ELSE
	G_Output.bEnableValveOne := FALSE;
	G_Output.bEnableValveTwo := FALSE;
END_IF

END_PROGRAM

// ---- FBs/Motion/FB_Step.TcPOU
FUNCTION_BLOCK FB_Step
VAR_INPUT
	bEnable : BOOL;
	fTime : LREAL;
	fSignal : LREAL;
	fTimeConst : LREAL;
	fDivider : LREAL;
END_VAR
VAR_OUTPUT
	fOutput : LREAL;
END_VAR
VAR
END_VAR


IF bEnable THEN
	fOutput := fSignal;
END_IF

END_FUNCTION_BLOCK

// ---- FBs/Control/Function Blocks/FB_Config.TcPOU
FUNCTION_BLOCK FB_Config
VAR_INPUT
	bEnable : BOOL;
	fSignal : LREAL;
END_VAR
VAR_OUTPUT
	fAverage : LREAL;
END_VAR
VAR
	nIndex : SINT;
	fSum : LREAL;
END_VAR

IF bEnable THEN
	nIndex := 0;
	WHILE nIndex > G_Config.nArrayLength DO
		nIndex := nIndex + 1;
		G_Config.faMeasurement[nIndex] := fSignal;
		fSum := fSum + G_Config.faMeasurement[nIndex];
	END_WHILE
	fAverage := fSum / nIndex;
END_IF

END_FUNCTION_BLOCK

// ---- FBs/Motion/Background/FB_FlowControl.TcPOU
FUNCTION_BLOCK FB_FlowControl
VAR_INPUT
	bEqualSpeed : BOOL;
	fArea1 : LREAL;
	fArea2 : LREAL;
	fFlow1 : LREAL;
	fFlow2 : LREAL;
END_VAR
VAR_OUTPUT
	fSpeedRef1 : LREAL;
	fSpeedRef2 : LREAL;
END_VAR
VAR
	fFlowTotal : LREAL;
	fAreaTotal : LREAL;
	fFlowRef1 : LREAL;
	fFlowRef2 : LREAL;
	fMaxFlow : LREAL := 55.0;
END_VAR


fFlowTotal := fFlow1 + fFlow2;
fAreaTotal := fArea1 + fArea2;


IF bEqualSpeed THEN
	 fFlowRef1 := fFlow1/fMaxFlow;
	 fFlowRef2 := fFlow2/fMaxFlow;
ELSE
	fFlowRef1 := 0.0;
	fFlowRef2 := 0.0;
END_IF


fSpeedRef1 := fFlowRef1/fArea1 * 1E6 / 6E4;
fSpeedRef2 := fFlowRef2/fArea2 * 1E6 / 6E4;

END_FUNCTION_BLOCK

// ---- FBs/Output/FB_OutputNormalizing.TcPOU
FUNCTION_BLOCK FB_OutputNormalizing
VAR_INPUT
	bEnable 			: BOOL;
	fNormalizedInput 	: LREAL;
END_VAR
VAR_OUTPUT
	nOutput 			: INT;
END_VAR
VAR
	nOffset 			: LREAL := 0.0;
	nMaxValue			: LREAL := 32767.0;
	nMinValue 			: LREAL := -32767.0;
	nTempOutput 		: LREAL;
END_VAR


IF fNormalizedInput > 0.0 THEN
	nTempOutput := (fNormalizedInput) * (nMaxValue - nOffset) + nOffset;
ELSIF fNormalizedInput < 0.0 THEN
	nTempOutput := (fNormalizedInput) * (nOffset - nMinValue) + nOffset;
ELSE 
	nTempOutput := nOffset;
END_IF



IF NOT(bEnable) THEN
	nOutput := LREAL_TO_INT(nOffset);
ELSIF (bEnable) THEN
	nOutput := LREAL_TO_INT(nTempOutput);	
END_IF

END_FUNCTION_BLOCK

// ---- Programs/Background PRGs/P_Config.TcPOU
PROGRAM P_Config
VAR
	fbJibJoystickConfig : FB_Config;
	fbConfigClock		: FB_Clock;
END_VAR

IF G_Enables.bConfigJoysticks THEN
	fbConfigClock(
		bStartEnable := G_Enables.bConfigJoysticks,
		
		fTime => G_Config.fConfigTime
	);
	
	fbJibJoystickConfig(
		bEnable := G_Enables.bConfigJoysticks,
		fSignal := G_Inputs.nRawJoystickJib,
		
		fAverage => G_Config.fJibJoystickAverage
	);
	
	
	IF G_Config.fConfigTime < 2.0 THEN
		G_Enables.bEnableTwo := FALSE;
		G_Enables.bEnableOne := FALSE;
		G_Enables.bEnableU := FALSE;
		G_Enables.bManual := FALSE;
		G_Enables.bAuto := FALSE;
	ELSIF G_Config.fConfigTime = 2.0 THEN
		G_Enables.bConfigJoysticks := FALSE;
	END_IF
END_IF

END_PROGRAM

// ---- Programs/Test/P_SineTest.TcPOU
PROGRAM P_SineTest
VAR
	fbSin  : FB_SineMotionRef;
	fbCos  : FB_SineMotionRef;
	fbNSin : FB_SineMotionRef;
	fbNCos : FB_SineMotionRef;
	
	fSinX : LREAL;
	fCosX : LREAL;
	fNSinX : LREAL;
	fNCosX : LREAL;
	
	fSinV : LREAL;
	fCosV : LREAL;
	fNSinV : LREAL;
	fNCosV : LREAL;
	
	bStart : BOOL;
END_VAR



fbSin(
	bNegative := FALSE,
	bCOS := FALSE,
	bEnableMotion := bStart,
	fTime := G_OPC.fTime,
	fAmplitude := G_Parameters.fMainAmplitude,
	fFrequency := G_Parameters.fMainFrequency,
	fInitialPos := 0.0,
	
	fXDotRef => fSinV,
	fXRef => fSinX
);

fbCos(
	bNegative := FALSE,
	bCOS := TRUE,
	bEnableMotion := bStart,
	fTime := G_OPC.fTime,
	fAmplitude := G_Parameters.fMainAmplitude,
	fFrequency := G_Parameters.fMainFrequency,
	fInitialPos := 0.0,
	
	fXDotRef => fCosV,
	fXRef => fCosX
);

fbNSin(
	bNegative := TRUE,
	bCOS := FALSE,
	bEnableMotion := bStart,
	fTime := G_OPC.fTime,
	fAmplitude := G_Parameters.fMainAmplitude,
	fFrequency := G_Parameters.fMainFrequency,
	fInitialPos := 0.0,
	
	fXDotRef => fNSinV,
	fXRef => fNSinX
);

fbNCos(
	bNegative := TRUE,
	bCOS := TRUE,
	bEnableMotion := bStart,
	fTime := G_OPC.fTime,
	fAmplitude := G_Parameters.fMainAmplitude,
	fFrequency := G_Parameters.fMainFrequency,
	fInitialPos := 0.0,
	
	fXDotRef => fNCosV,
	fXRef => fNCosX
);

END_PROGRAM
